// TwinCAT 3 PLC project Emulator
// ProgramVersion: 3.1.4024.12
// libraries:
//   Tc2_ModbusRTU, * (Beckhoff Automation GmbH)
//   Tc2_ModbusSrv, * (Beckhoff Automation GmbH)
//   Tc2_Standard, * (Beckhoff Automation GmbH)
//   Tc2_System, * (Beckhoff Automation GmbH)
//   Tc2_TcpIp, * (Beckhoff Automation GmbH)
//   Tc2_Utilities, * (Beckhoff Automation GmbH)
//   Tc3_Module, * (Beckhoff Automation GmbH)
// project tree:
//   00_FunctionsBlocks/AlarmManagement/ FB_AlarmCodeManager.TcPOU, FB_CheckCommand.TcPOU, FB_CheckSetpt.TcPOU, FB_DetectFixedValue.TcPOU, FB_DetectFlicker.TcPOU, FB_HeartBeatMasterBackup.TcPOU, FB_UnknownEvent.TcPOU, FUN_Alarms_CSV.TcPOU, FUN_ReadAlarm_CSV.TcPOU, ServerCSV.TcDUT, ServerSms.TcDUT, SMS_Server.TcPOU
//   00_FunctionsBlocks/Annexesfunction/ FUN_ConnectVPN.TcPOU, FUN_DisconnectVPN.TcPOU, FUN_GetPublicIp.TcPOU, FUN_PingHost.TcPOU, PRG_RestartPlc.TcPOU, PRG_RestartService.TcPOU
//   00_FunctionsBlocks/BoolManagement/ FB_CountNinTimeWindow.TcPOU, FB_TapVariable.TcPOU, FB_Toggle2Tap.TcPOU, FB_WordToArrayOfBool.TcPOU, FB_WriteOnChange.TcPOU, RS_NoReset.TcPOU
//   00_FunctionsBlocks/Communication/IEC104/ E_ComState.TcDUT, FB_IEC104ServerAkuo.TcPOU, GVL_Cst.TcGVL, ST_IEC104AkuoParam.TcDUT
//   00_FunctionsBlocks/Communication/Mail/ FUN_SendMail.TcPOU, ServerMail.TcDUT
//   00_FunctionsBlocks/Communication/ModbusRTU/ CheckStruct.TcPOU, FB_ModbusRTU.TcPOU, FB_ReadModbusRTU_V2.TcPOU, Sample_ModbusRTU.TcPOU, Struct_InputRTU.TcDUT
//   00_FunctionsBlocks/Communication/ModbusTCP/ FB_ModbusRead.TcPOU, FB_ModbusReadCoils.TcPOU, FB_ModbusReadInput.TcPOU, FB_ModbusReadInputRegs.TcPOU, FB_ModbusWrite.TcPOU, FB_ModbusWriteMultipleCoils.TcPOU, FB_ModbusWriteSingleCoil.TcPOU, FB_ModbusWriteSingleRegister.TcPOU
//   00_FunctionsBlocks/Communication/SMS/ FB_DeleteAllSMS.TcPOU, FB_DeleteSMS.TcPOU, FB_Extract_Num_Mes.TcPOU, FB_Login.TcPOU, FB_ReadSMS.TcPOU, FB_SendSMS.TcPOU, ST_SMSDataSetEntry_Read.TcDUT, ST_SMSDataSetEntry_Send.TcDUT
//   00_FunctionsBlocks/Ctrl/ FB_PIDRegulation.TcPOU
//   00_FunctionsBlocks/Database/ CheckConfig.TcPOU, PRG_EpochConverter.TcPOU, PRG_TimestructConverter.TcPOU, St_DataHisto.TcDUT, St_DataHisto_Epoch.TcDUT, UnixTimestamp.TcPOU
//   00_FunctionsBlocks/Database/Firebird/ Firebird_CreateTables.TcPOU, Firebird_InsertBuffer.TcPOU, Firebird_InsertBuffer_vEpoch.TcPOU, Firebird_ReadAlarms.TcPOU, Firebird_RetrieveHDBID.TcPOU, Firebird_SelectBuffer.TcPOU, Firebird_WriteAlarms.TcPOU, LoggerFirebird.TcDUT, St_AlarmsV2.TcDUT
//   00_FunctionsBlocks/Database/InfluxDb/ InfluxDb_AlarmsManagement.TcPOU, InfluxDb_ReadValues.TcPOU, InfluxDb_WriteAlarms.TcPOU, InfluxDb_WriteStruct.TcPOU, LoggerInfluxDb.TcDUT, ST_InfluxAlarmsInsert.TcDUT, ST_InfluxAlarmsRetrieve.TcDUT
//   00_FunctionsBlocks/Database/SQLCe/ FB_SQLExpert_InsertBuffer_1.TcPOU
//   00_FunctionsBlocks/Database/SQLite/ SQLite_CreateDb_V2_1.TcPOU, SQLite_DeleteConfDb_1.TcPOU
//   00_FunctionsBlocks/DataProcessing/Compress/ FB_CompressFile.TcPOU, FUN_CompressCSV.TcPOU
//   00_FunctionsBlocks/DataProcessing/Database/ DataBase_V2.TcPOU, FB_DeleteFile.TcPOU, FB_SQLExpert_InsertBuffer.TcPOU, SQLite_CreateDb_V2.TcPOU, SQLite_DeleteConfDb.TcPOU
//   00_FunctionsBlocks/DataProcessing/ FB_Average.TcPOU, FB_CountBitOfWordAtTrue.TcPOU, FB_Integrate.TcPOU, FB_MessageDynamique.TcPOU, FB_MovingAverage.TcPOU, FB_Ramp.TcPOU, FB_Ramp_Time.TcPOU, FB_Smooth.TcPOU, FB_XorWord.TcPOU, FUN_Transpose.TcPOU, ReplaceAll.TcPOU, SavePersistent.TcPOU, Split.TcPOU, Substring.TcPOU
//   00_FunctionsBlocks/DataProcessing/MergeWord/ FB_ISKRA_T5.TcPOU, FB_ISKRA_T6.TcPOU, FB_MergeWordsToDint.TcPOU, FB_MergeWordsToFloat.TcPOU, FB_MergeWordsToUint.TcPOU, FB_MergeWordsToUlint.TcPOU, FB_SplitFloatToWords.TcPOU, FB_WordsToDint64BE.TcPOU, FB_WordsToFloat32MLE.TcPOU
//   00_FunctionsBlocks/DataProcessing/ReadFile/ FB_Read.TcPOU, FB_ReadCSV.TcPOU
//   00_FunctionsBlocks/DataProcessing/SplitWord/ FB_SplitRealToWords.TcPOU, FB_SplitRealToWords_IEEE754.TcPOU, FB_SplitUlintToWords.TcPOU, FB_SplitWordToByte.TcPOU
//   00_FunctionsBlocks/DataProcessing/WriteFile/ CheckStruct_Alarms.TcPOU, FB_CreateDir_V2.TcPOU, FB_WriteFile.TcPOU, FB_Write_CSV.TcPOU, FUN_CreateDir_CSV.TcPOU, LoggerCSV.TcDUT, ST_Journal.TcDUT, ST_ValuesAlarms.TcDUT, ST_ValuesWrite.TcDUT
//   00_FunctionsBlocks/Fifo/ FB_CommandAlternate.TcPOU, FB_DBDatasetFifo.TcPOU, FB_DBDatasetFifo_1min.TcPOU, FB_SMSDatasetFifo_Read.TcPOU, FB_SMSDatasetFifo_Send.TcPOU, GVL_Fifo.TcGVL
//   00_FunctionsBlocks/HistorizationVisu/ FB_OperationIndex.TcPOU, GetTime.TcPOU
//   00_FunctionsBlocks/Templates/ FB_EX_Example.TcPOU
//   01_Equipement_Library/Actuators/ CB_AuxMVCB_Sch.TcDUT, CB.TcDUT, CB_Standard.TcDUT, FB_CB_AuxMVCB.TcPOU, FB_CB_Base.TcPOU, FB_CB_FeederMVCB.TcPOU, FB_CB_GridMVCB.TcPOU, FB_CB_MainHVCB.TcPOU, FB_CB_MainMVCB.TcPOU, FB_CB_MeasureMVCB.TcPOU, FB_CB_MVSwitch.TcPOU, CB_FeederMVCB_Sch.TcDUT, CB_MainHVCB_Sch.TcDUT, CB_MainMVCB_Sch.TcDUT, CB_MeasureMVCB_Sch.TcDUT
//   01_Equipement_Library/Batteries/ Cell.TcDUT, FB_SystemBMS_Base.TcPOU, FB_SystemBMS_M3.TcPOU, Rack.TcDUT, RackString.TcDUT, SystemBMS.TcDUT
//   01_Equipement_Library/Datalogger/ Datalogger.TcDUT, Datalogger_PPCVerrerie.TcDUT, Datalogger_SchSkid.TcDUT, Datalogger_SENECA.TcDUT, FB_Datalogger_Base.TcPOU, FB_Datalogger_PPCVerrerie.TcPOU, FB_Datalogger_SchSkid.TcPOU, FB_Datalogger_SENECA.TcPOU
//   01_Equipement_Library/Fan/ Fan.TcDUT, FB_Fan_Basic.TcPOU
//   01_Equipement_Library/FireSystem %28FSS%29/ FB_FSS.TcPOU (not stored), FSS.TcDUT (not stored), FSS_Standard.TcDUT (not stored)
//   01_Equipement_Library/GRID/ FB_GRID_Base.TcPOU, FB_GRID_Enedis.TcPOU, GRID.TcDUT, GRID_Enedis.TcDUT
//   01_Equipement_Library/HVAC/ FB_HVAC.TcPOU, FB_HVAC_Base.TcPOU, FB_HVAC_MADI.TcPOU, FB_HVAC_Standard.TcPOU, HVAC.TcDUT, HVAC_MADI.TcDUT, HVAC_Standard.TcDUT
//   01_Equipement_Library/Inverter/ FB_INV_1000CP_XT.TcPOU, FB_INV_Base.TcPOU, FB_INV_Sch4400.TcPOU, FB_INV_Smartlogger.TcPOU, FB_INV_Sun2000KtlMo.TcPOU, INV.TcDUT, INV_1000CP_XT.TcDUT, INV_1000CP_XT_StringMonitor.TcDUT, INV_Huawei.TcDUT, INV_Sch4400.TcDUT, SL_Huawei.TcDUT, STR.TcDUT
//   01_Equipement_Library/IPC/ FB_IPC.TcPOU, IPC.TcDUT
//   01_Equipement_Library/Operation Meter/ FB_PM_520_230.TcPOU, FB_PM_A40.TcPOU, FB_PM_Base.TcPOU, FB_PM_ION7650.TcPOU, FB_PM_Janitza.TcPOU, FB_PM_PM3250.TcPOU, FB_PM_PM800.TcPOU, FB_PM_SicamQ100.TcPOU, FB_PM_SM103E.TcPOU, PM.TcDUT, PM_PM800.TcDUT, PM_Q100.TcDUT, PM_SicamQ100.TcDUT, PM_Standard.TcDUT
//   01_Equipement_Library/PCS/ FB_PCS_Base.TcPOU, FB_PCS_Jema.TcPOU, PCS.TcDUT, PowerCol_Jema.TcDUT, PowerCol_Jema_Alarms.TcDUT
//   01_Equipement_Library/ProtectRelay/ FB_ProtectRelay_Base.TcPOU, FB_ProtectRelay_DM2.TcPOU, FB_ProtectRelay_Flair23DM.TcPOU, FB_ProtectRelay_NSXCB.TcPOU, FB_ProtectRelay_PACE100ST.TcPOU, FB_ProtectRelay_REF615.TcPOU, FB_ProtectRelay_SEPAM10a.TcPOU, FB_ProtectRelay_SepamS48.TcPOU, FB_ProtectRelay_SepamT20.TcPOU, FB_ProtectRelay_VIP410.TcPOU, FB_ProtectRelay_WIP1.TcPOU, ProtectRelay.TcDUT, ProtectRelay_Flair23DM.TcDUT, ProtectRelay_NSXCB.TcDUT, ProtectRelay_PACE100ST.TcDUT, ProtectRelay_REFIO.TcDUT, ProtectRelay_S42.TcDUT, ProtectRelay_S48.TcDUT, ProtectRelay_T20.TcDUT, ProtectRelay_T87.TcDUT, ProtectRelay_VIP410.TcDUT, ProtectRelay_WIP1.TcDUT
//   01_Equipement_Library/Router/ FB_Router.TcPOU, Router.TcDUT, Router_Standard.TcDUT
//   01_Equipement_Library/Sensors/ANA/ ANA.TcDUT, FB_ANA_Base.TcPOU, FB_ANA_IO.TcPOU, FB_ANA_Irra_Fx.TcPOU
//   01_Equipement_Library/Sensors/COM/ AllInOne.TcDUT, FB_AllInOne.TcPOU, FB_ANA_SMP1X.TcPOU, SMP1X.TcDUT
//   01_Equipement_Library/Sensors/TOR/ FB_TOR_Base.TcPOU, FB_TOR_CB.TcPOU, FB_TOR_DS.TcPOU, FB_TOR_ES.TcPOU, FB_TOR_Fuse.TcPOU, FB_TOR_MS.TcPOU, FB_TOR_Rain.TcPOU, FB_TOR_SD.TcPOU, FB_TOR_Spd.TcPOU, FB_TOR_Standard.TcPOU, FB_TOR_ToS.TcPOU, TOR.TcDUT, TOR_Rain.TcDUT, TOR_Standard.TcDUT
//   01_Equipement_Library/Tariff Meter/ EM.TcDUT, EM_Standard.TcDUT, FB_EM.TcPOU, FB_EM_Base.TcPOU, FB_EM_Pulse.TcPOU
//   01_Equipement_Library/Transfo/ FB_Transfo_Base.TcPOU, FB_Transfo_HVCom.TcPOU, FB_Transfo_MV.TcPOU, FB_Transfo_MVCom.TcPOU, Transfo.TcDUT, Transfo_HV.TcDUT, Transfo_MV.TcDUT
//   01_Equipement_Library/UPS/ FB_UPS_Base.TcPOU, FB_UPS_CXC.TcPOU, FB_UPS_Eneris.TcPOU, FB_UPS_PS10048.TcPOU, UPS.TcDUT, UPS_CXC.TcDUT, UPS_ENERIS.TcDUT, UPS_Eneris.TcDUT, UPS_Eneris.TcDUT, UPS_PS10048.TcDUT
//   02_Product_Library/EnergyStorageSystem%28ESS%29/ ESS.TcDUT (not stored), FB_ESS.TcPOU (not stored), FB_ESS_Base.TcPOU (not stored)
//   02_Product_Library/PowerTRansformerStation%28PTR%29/ FB_PTR.TcPOU (not stored), FB_PTR_Base.TcPOU (not stored), PTR.TcDUT (not stored), PTR_Exd.TcDUT (not stored)
//   02_Product_Library/Substation%28SUB_HV%29/ FB_SUBHV.TcPOU (not stored), FB_SUBHV_Base.TcPOU (not stored), SUBHV.TcDUT (not stored), SUBHV_Exd.TcDUT (not stored)
//   02_Product_Library/Substation%28SUB_MV%29/ FB_SUBMV.TcPOU (not stored), FB_SUBMV_Base.TcPOU (not stored), SUBMV.TcDUT (not stored), SUBMV_Exd.TcDUT (not stored)
//   02_Product_Library/WeatherStation %28WS%29/ FB_WS.TcPOU (not stored), FB_WS_Base.TcPOU (not stored), WS.TcDUT (not stored), WS_AGMA.TcDUT (not stored)
//   03_Power_Plant %28PP%29/ FB_PP.TcPOU (not stored), PP.TcDUT (not stored)
//   04_Application/ADS/ ADS_Custom.TcPOU, ADS_Param.TcPOU
//   04_Application/Checks/ CheckBounds.TcPOU, CheckDivDInt.TcPOU, CheckDivLInt.TcPOU, CheckDivLReal.TcPOU, CheckDivReal.TcPOU, CheckLRangeSigned.TcPOU, CheckLRangeUnsigned.TcPOU, CheckPointer.TcPOU, CheckRangeSigned.TcPOU, CheckRangeUnsigned.TcPOU
//   04_Application/CONFIG/ GVL_BASE.TcGVL, GVL_Beckhoff.TcGVL, GVL_CFG.TcGVL, GVL_Check.TcGVL, GVL_DataBaseStructures.TcGVL, GVL_EmulConfig.TcGVL
//   04_Application/IO/ IO.TcDUT, PRG_IO.TcPOU, ST_AI.TcDUT, ST_AO.TcDUT, ST_DI.TcDUT, ST_DO.TcDUT
//   04_Application/MAIN/ MAIN_Emul.TcPOU
//   / Emul_Task.TcTTO

CONFIGURATION Emulator
    RESOURCE PLC ON TwinCAT3
        TASK Emul_Task(INTERVAL := T#25000us, PRIORITY := 16);
        PROGRAM MAIN_Emul WITH Emul_Task : MAIN_Emul;
    END_RESOURCE
END_CONFIGURATION

// ---- 00_FunctionsBlocks/AlarmManagement/ServerCSV.TcDUT

TYPE ServerCSV :
STRUCT
	FileSize			: ULINT;			(*(o) Size of the file being used for logging alarms *)
	TimeCreation		: TIMESTRUCT;		(* TimeCreation of file*)
	TimeModif			: TIMESTRUCT;		(* Time Modif of file*)
	MesAlarmCode		: WORD;				(* Alarm Code related to this functionnality*)

END_STRUCT
END_TYPE

// ---- 00_FunctionsBlocks/AlarmManagement/ServerSms.TcDUT

TYPE ServerSms :
STRUCT
	NbrUtiliActive			: INT;									(* Number of users*)
	MesAlarmCode			: WORD;									(* Alarm Code*)
	AX_Numtel				: ARRAY[1..CstNbUser] OF STRING(26);	(*Tel Number list*)
	AX_Subscribed			: ARRAY[1..CstNbUser] OF BOOL;			(*Subscription list*)
	AX_NomUtili				: ARRAY[1..CstNbUser] OF STRING(50); 	(* User name list	*)
	AX_UserLVL				: ARRAY[1..CstNbUser] OF WORD; 		(*User Level*)

END_STRUCT
END_TYPE

// ---- 00_FunctionsBlocks/Communication/IEC104/E_ComState.TcDUT
TYPE E_ComState :
(
	INIT := 0,
	IDLE,
	CONNECT,
	DATATRANSFER,
	DISCONNECT
);
END_TYPE

// ---- 00_FunctionsBlocks/Communication/IEC104/ST_IEC104AkuoParam.TcDUT
TYPE ST_IEC104AkuoParam :
STRUCT
	bEnableFlicker 	: BOOL :=  TRUE ;
	tFlickerWindow	: TIME := T#10S ; 
	uFlickerNumber	: UINT := 7  ; 

	iLocalPort 		: UDINT := 2404;						// locl port
	sLocalHost		: STRING := '127.0.0.1'; 			// server IP address. 
	iAOnb			: INT ;								// Number of AO being treated ( <GVL_Cst.CstNbAOEntries)
 
END_STRUCT
END_TYPE

// ---- 00_FunctionsBlocks/Communication/Mail/ServerMail.TcDUT

TYPE ServerMail :
STRUCT

	MesAlarmCode			: WORD;			(*alarm code *)
	
	AX_MailAddr				: ARRAY[1..CstNbUser] OF STRING(255);		(* Mail Address List*)
	AX_Subscribed			: ARRAY[1..CstNbUser] OF BOOL;				(* Mail subscription list*)
	AX_NomUtili				: ARRAY[1..CstNbUser] OF STRING(50); 		(* User Name List*)
	AX_UserLVL				: ARRAY[1..CstNbUser] OF WORD; 		(* User Level*)
	
	OUT_NbMailSent			: ULINT;									(* Number of mail being sent *)
	
END_STRUCT
END_TYPE

// ---- 00_FunctionsBlocks/Communication/ModbusRTU/Struct_InputRTU.TcDUT
TYPE Struct_InputRTU :
STRUCT
	InStartAddr			: WORD;
	InQuantity			: WORD;
	InUnitID			: BYTE;
	InBuffer			: POINTER TO BYTE;
	InFunction			: UINT;
	OutBusy				: POINTER TO BOOL;
	OutError			: POINTER TO BOOL;
	OutCompleted 		: POINTER TO BOOL;
	OutErrorId			: POINTER TO INT ; 
END_STRUCT
END_TYPE

// ---- 00_FunctionsBlocks/Communication/SMS/ST_SMSDataSetEntry_Read.TcDUT
TYPE ST_SMSDataSetEntry_Read :
STRUCT
	Message : STRING(160);  // Commande envoyé par message
	Num		: STRING(20);  //  Numéro de l'utilisateur
END_STRUCT
END_TYPE

// ---- 00_FunctionsBlocks/Communication/SMS/ST_SMSDataSetEntry_Send.TcDUT
TYPE ST_SMSDataSetEntry_Send :
STRUCT
	ID				: UINT;			// Unic ID to identify the alarm
	IndexWord		: UINT; 		//Index du word correspondant aux alarmes
	IndexBit		: UINT; 		//Index du bit correspondant a l'alarme
	Active			: BOOL; 		//Ne pas remplir - Utilisé par le code
	Num_tel			: STRING(20);//Ne pas remplir - Utilisé par le code
	TimeStamp_Act	: STRING;	// TimeStamp of the last activation or desactivation
	Alarms_LVL		: WORD;
END_STRUCT
END_TYPE

// ---- 00_FunctionsBlocks/Database/Firebird/LoggerFirebird.TcDUT

TYPE LoggerFirebird :
STRUCT
	MesAlarmCode		: WORD;				// Alarm Code

END_STRUCT
END_TYPE

// ---- 00_FunctionsBlocks/Database/Firebird/St_AlarmsV2.TcDUT
TYPE St_AlarmsV2 :
STRUCT
	TIMESTAMP_START : DT;
	TIMESTAMP_STOP	: DT;
	ALARMSID 		: DINT;
	ACT				: INT;
	ACK				: INT;
	

END_STRUCT
END_TYPE

// ---- 00_FunctionsBlocks/Database/InfluxDb/LoggerInfluxDb.TcDUT
TYPE LoggerInfluxDb :
STRUCT
	MesAlarmCode		: WORD;				// Alarm Code
END_STRUCT
END_TYPE

// ---- 00_FunctionsBlocks/Database/InfluxDb/ST_InfluxAlarmsInsert.TcDUT
TYPE ST_InfluxAlarmsInsert :
STRUCT
    {attribute 'TagName' := 'Message'}
	Message		 	: T_MaxString;	// Alarm Message 
    {attribute 'FieldName' := 'ID'}	
	ID			: 	ULINT;
    {attribute 'FieldName' := 'Value'}	
	Value 		: BOOL;
    {attribute 'FieldName' := 'Ack'}	
	Ack			: BOOL;	
END_STRUCT
END_TYPE

// ---- 00_FunctionsBlocks/Database/InfluxDb/ST_InfluxAlarmsRetrieve.TcDUT
TYPE ST_InfluxAlarmsRetrieve :
STRUCT
    {attribute 'TagName' := 'time'}
	MesTime			: LINT;
    {attribute 'TagName' := 'Message'}
	Message		 	: T_MaxString;	// Alarm Message 
    {attribute 'FieldName' := 'ID'}	
	ID				: ULINT;
    {attribute 'FieldName' := 'Value'}	
	Value 			: BOOL;
    {attribute 'FieldName' := 'Ack'}	
	Ack				: BOOL;	
END_STRUCT
END_TYPE

// ---- 00_FunctionsBlocks/Database/St_DataHisto.TcDUT
TYPE St_DataHisto :
STRUCT
	Timestamp		: TIMESTRUCT;
	ParentId		: DINT;
	Value			: LREAL;
END_STRUCT
END_TYPE

// ---- 00_FunctionsBlocks/Database/St_DataHisto_Epoch.TcDUT
TYPE St_DataHisto_Epoch :
STRUCT
	Timestamp		: ULINT;
	ParentId		: DINT;
	Value			: LREAL;
END_STRUCT
END_TYPE

// ---- 00_FunctionsBlocks/DataProcessing/WriteFile/LoggerCSV.TcDUT

TYPE LoggerCSV :
STRUCT
	FileSize			: ULINT;			(* (o) File size *)
	TimeCreation		: TIMESTRUCT;		(* TimeCreation of file*)
	TimeModif			: TIMESTRUCT;		(* Time Modif of file*)
	MesAlarmCode		: WORD;				(* Alarm Code*)

END_STRUCT
END_TYPE

// ---- 00_FunctionsBlocks/DataProcessing/WriteFile/ST_Journal.TcDUT
TYPE ST_Journal :
STRUCT
	Message			: STRING(150); //Message texte à envoyer aux utilisateurs
	Groupe			: (Sans_Operation,Avec_Operation_Act,Avec_Operation_Act_Des):=1; // 0:sans action,1:Envois sms sur acttivation,2:Envois sms sur activation et desactivation
	Ax_ParamB		: ARRAY [1..4] OF POINTER TO BOOL; //Tableau boolean permettant d'envoyer un message dynamique.
	Ax_ParamI		: ARRAY [1..4] OF POINTER TO SINT; //Tableau Sint permettant d'envoyer un message dynamique.
END_STRUCT
END_TYPE

// ---- 00_FunctionsBlocks/DataProcessing/WriteFile/ST_ValuesAlarms.TcDUT
TYPE ST_ValuesAlarms :
STRUCT
	ID				: UINT;		// Unic ID to identify the alarm 
	Message		 	: STRING(160);	// Alarm Message 
	Value 			: BOOL;		// Value of the alarm
	Ack 			: BOOL;		// Ack of the alarm	
	TimeStamp_Act	: STRING;	// TimeStamp of the last activation or desactivation
	
	Groupe			: UINT:=0; // 0:sans action,1:Envois sms sur acttivation,2:Envois sms sur activation et desactivation
	Alarms_LVL		: WORD:=1; // Si Num utilisateur > Alarms_LVL alors il ne recoit pas les sms 1 := Standart , 2 := Syntehses , 3:= Securité
END_STRUCT
END_TYPE

// ---- 00_FunctionsBlocks/DataProcessing/WriteFile/ST_ValuesWrite.TcDUT
TYPE ST_ValuesWrite :
STRUCT
	Description : STRING;
	Address 	: POINTER TO REAL;
	AddressLR	: POINTER TO LREAL;
	AddressUL	: POINTER TO ULINT;
	AddressUI	: POINTER TO UINT;
	Size		: UINT;
	Sampling	: DINT := 1000;		// Period of sampling
	
END_STRUCT
END_TYPE

// ---- 01_Equipement_Library/Actuators/CB_AuxMVCB_Sch.TcDUT
///////////
// Structure For Bousquet. Main Operating Data to be saved (ex: OPC).  
//////////

TYPE CB_AuxMVCB_Sch :
STRUCT
	//DI
	MesData					: CB ;      (* Object*)
	MesFuseBurned		    : BOOL ; 	(* The Fuse is burned*)
	MesEarth				: BOOL ; 	(* The Cell is grounded*)

END_STRUCT
END_TYPE

// ---- 01_Equipement_Library/Actuators/CB.TcDUT
TYPE CB :
///////////
// Structure For Bousquet. Main Operating Data to be saved ( ex: OPC )   
//////////
STRUCT
	//DI
	MesClosed		: BOOL ;	(* Cell is closed*)
	MesOpened		: BOOL ;	(* cell is opened*)
	
	MesAlarmCode	: WORD ;	(* Internal Akuo Alarm Code*)
	MesWarningCode	: WORD ;	(* Internal Akuo Warning Code*)
	MesEventCode	: WORD ;	(* Internal Akuo Warning Code*)
	
	MesCP_Open		: BOOL ;   	(* Cal(NA) Permanent Conditions*)
	MesCP_Close		: BOOL ; 	(* Cal(NA) Permanent Conditions*) 

END_STRUCT
END_TYPE

// ---- 01_Equipement_Library/Actuators/CB_Standard.TcDUT
TYPE CB_Standard :
///////////
// Structure For Bousquet. Main Operating Data to be saved ( ex: OPC )   
//////////
STRUCT
	//DI
	MesData				: CB ;  (* Object*)

END_STRUCT
END_TYPE

// ---- 01_Equipement_Library/Actuators/CB_FeederMVCB_Sch.TcDUT
///////////
// Structure For Bousquet . Main Operating Data to be saved (ex: OPC).  
//////////

TYPE CB_FeederMVCB_Sch :
STRUCT
	//DI
	MesData					: CB   ;    (* Object*)
	MesComutLocal		    : BOOL ; 	(* The cell selector is in local position*)
	MesAlarmPwr		        : BOOL ; 	(* The cell motorization has a power supply fault*)
	MesEarth				: BOOL ; 	(* The cell is grounded (earthing)*)
	MesTripped	    	    : BOOL ; 	(* The cell is tripped (opened and locked due to alarm)*)
	OUT_CmdOpen				: BOOL ; 	(* The SCADA sends an Open command to the cell*)
	OUT_CmdClose			: BOOL ; 	(* The SCADA sends a Close command to the cell*)
	MesOpened_Sect			: BOOL ;    (* The associated switchgear is opened*)
	
END_STRUCT
END_TYPE

// ---- 01_Equipement_Library/Actuators/CB_MainHVCB_Sch.TcDUT
///////////
// Structure For Bousquet . Main Operating Data to be saved (ex: OPC).  
//////////

TYPE CB_MainHVCB_Sch :
STRUCT
	//DI
	MesData					: CB   ;    (* Object*)
	MesComutLocal		    : BOOL ; 	(* The cell selector is in local position*)
	MesAlarmPwr		        : BOOL ; 	(* The cell motorization has a power supply fault*)
	MesEarth				: BOOL ; 	(* The cell is grounded (earthing)*)
	MesTripped	    	    : BOOL ; 	(* The cell is tripped (opened and locked due to alarm)*)

	MesAlarm_SF6      			: BOOL ; (* Not enough SF6 gaz *)
	MesAlarm_Disarmed      		: BOOL ; (* HVCB Command is disarmed*)
	MesAlarm_ArmingMotor   		: BOOL ; (* Arming motorization is on fault*)
	MesAlarm_230V  		 		: BOOL ; (* 230V Aux is on fault*)
	MesOpened_Sect				: BOOL ; (* The associated switchgear is opened*)
	
END_STRUCT
END_TYPE

// ---- 01_Equipement_Library/Actuators/CB_MainMVCB_Sch.TcDUT
///////////
// Structure for MainMVCB Schneider. Main Operating Data to be saved (ex: OPC).  
//////////

TYPE CB_MainMVCB_Sch :
STRUCT
	//DI
	MesData					: CB   ;    (* Object*)
	MesComutLocal		    : BOOL ; 	(* The cell selector is in local position*)
	MesAlarmPwr		        : BOOL ; 	(* The cell motorization has a power supply fault*)
	MesEarth				: BOOL ; 	(* The cell is grounded (earthing)*)
	MesTripped	    	    : BOOL ; 	(* The cell is tripped (opened and locked due to alarm)*)
	OUT_CmdOpen				: BOOL ; 	(* The SCADA sends an Open command to the cell*)
	OUT_CmdClose			: BOOL ; 	(* The SCADA sends a Close command to the cell*)
	MesOpened_Sect			: BOOL ; 	(* The associated switchgear is opened*)
	
END_STRUCT
END_TYPE

// ---- 01_Equipement_Library/Actuators/CB_MeasureMVCB_Sch.TcDUT
///////////
// Structure For Bousquet. Main Operating Data to be saved (ex: OPC).  
//////////

TYPE CB_MeasureMVCB_Sch :
STRUCT
	//DI
	MesData					: CB ;      (* Object*)
	MesFuseBurned		    : BOOL ; 	(* The Fuse is burned*)
	MesEarth				: BOOL ; 	(* The Cell is grounded*)

END_STRUCT
END_TYPE

// ---- 01_Equipement_Library/Batteries/Cell.TcDUT
///////////
// Structure For Battery Racks. Main Operating Data to be saved ( ex: OPC ) .  
//////////
TYPE Cell :
STRUCT
	MesU			: REAL ;    		(*( V) Cell voltage *)
	
END_STRUCT
END_TYPE

// ---- 01_Equipement_Library/Batteries/Rack.TcDUT
///////////
// Structure For Battery Racks. Main Operating Data to be saved ( ex: OPC ) .  
//////////
TYPE Rack :
STRUCT
	
		// Info of Rack BBMS  
		ParamNbStrings			: UINT ; 	// 		Number of strings for the rack set in BBMS 
		MesHeartBeat			: UINT;		// (NA) Rack's Heartbeat, increases by 1 every second
		MesAlarm1				: WORD;		// (NA) bit0: 
		MesAlarm2				: WORD;		// (NA) bit0: 
		MesProtection1			: WORD;		// (NA) bit0: 
		MesProtection2			: WORD;		// (NA) bit0: 		
		MesSwitchControlStatus	: WORD ; 	// Control status
		MesSwitchSensorStatus	: WORD ; 	// Sensor status
		MesUSwtchGrPackPlus		: REAL;		// (V)	a measured value of voltage applied to pack(+) of switchgear
		MesTempPCB				: REAL ; 	// (°C) Temperature Rack PCB 
		MesIdcFaultLvl			: UINT ;	//		Current Level when power is cut (1/2/3/4/5/6/7/8/9/10 : 1200A/700A/500A/200A/0A/-0A/-200A/-500A/-700A/-1200A)
		MesDcOpenCount			: UINT ; 	// Count number of dc opening 
		MesDcCloseCount			: UINT ; 	// Count number of dc closing 
		
		AX_RACKSTRING			: ARRAY[1..1] OF RackString ; 	// object 
	
		CalRackClosed			: BOOL ; 		// Rack ( Main DC contactor )is closed 

END_STRUCT
END_TYPE

// ---- 01_Equipement_Library/Batteries/RackString.TcDUT
///////////
// Structure For Battery Racks. Main Operating Data to be saved ( ex: OPC ) .  
//////////
TYPE RackString :
STRUCT
	
		MesMode								: UINT;		// (NA) Rack mode: 0: None, 1: Init, 2: Off, DcSwitch On, 3: On, DcSwitch On,
		MesAlarm1							: WORD;		// (NA) bit0: 
		MesAlarm2							: WORD;		// (NA) bit0: 
		MesAlarm3							: WORD;		// (NA) bit0: 
		MesAlarm4							: WORD;		// (NA) bit0: 
		MesProtection1						: WORD;		// (NA) bit0: 
		MesProtection2						: WORD;		// (NA) bit0: 
		MesProtection3						: WORD;		// (NA) bit0: 
		MesProtection4						: WORD;		// (NA) bit0: 		
		MesControlStatus					: WORD ; 	// Control Status
		MesUdc								: REAL ; 	// String Voltage 
		MesUdc_ModuleSum					: REAL  ;	// String voltage obtained by summing module voltage 
		MesUdc_CellSum						: REAL ; 	// String voltage obtained by summing Cell voltage 
		MesIdc								: REAL;		// (A) Rack Current
		MesIdc_Avg							: REAL;		// (A) Rack Current ( average of 3 sec) 
		MesSoC	 							: REAL;  	// (%) SoC on Battery rack 
		MesSoH	 							: REAL;  	// (%) SoH on Battery rack 
		MesCCL								: REAL;		// (A) Charge limit of rack
		MesDCL								: REAL;		// (A) Discharge limit of rack
		MesCPL								: REAL ; 	// (kW) Charge Power Limit		- To zero if Estop is set . 
		MesDPL								: REAL ; 	// (kW) Discharge Power Limit - To zero if Estop is set .
		MesECharge							: REAL ; 	// (kWh) Total Energy charged over time 
		MesEDischarge						: REAL ; 	// (kWh) Total Energy Discharge over time 
		MesOff_ModuleID						: UINT; 	// Module ID where the power is off while the other modules are connected . 
		MesComError_ModuleID				: UINT ; 	// Module ID where there is a LOC while other modules are connected . 
		MesUdcDiffMax_Cell					: REAL ; 	// (V) 	Max voltage difference between cells . 
		MesUdc_Cell							: REAL; 	// (V)	Cell voltage. Average
		MesUdcMax1_Cell						: REAL; 	// (V)	Cell voltage. Max Rank #1
		MesUdcMax1_Cell_ModuleID			: UINT; 	// (V)	Module ID where Cell voltage  reaches Max value. Rank #1
		MesUdcMax1_Cell_CellID				: UINT; 	// (V)	Cell ID where Cell voltage reaches Max value. Rank #1
		MesUdcMin1_Cell						: REAL; 	// (V)	Cell voltage . Min Rank #1
		MesUdcMin1_Cell_ModuleID			: UINT; 	// (V)	Module ID where Cell voltage  reaches Min value. Rank #1
		MesUdcMin1_Cell_CellID				: UINT; 	// (V)	Cell ID where Cell voltage reaches Min value. Rank #1
		MesUdcMax2_Cell						: REAL; 	// (V)	Cell voltage . Max Rank #2
		MesUdcMax2_Cell_ModuleID			: UINT; 	// (V)	Module ID where Cell voltage  reaches Max value. Rank #2
		MesUdcMax2_Cell_CellID				: UINT; 	// (V)	Cell ID where Cell voltage reaches Max value. Rank #2
		MesUdcMin2_Cell						: REAL; 	// (V)	Cell voltage . Min Rank #2
		MesUdcMin2_Cell_ModuleID			: UINT; 	// (V)	Module ID where Cell voltage  reaches Min value. Rank #2
		MesUdcMin2_Cell_CellID				: UINT; 	// (V)	Cell ID where Cell voltage reaches Min value. Rank #2		
		MesTempDiffMax_Cell					: REAL ; 	// (°C) Max Temp difference between cells . 
		MesTemp_Cell						: REAL; 	// (°C)	Cell Temp . Average
		MesTempMax1_Cell					: REAL; 	// (°C)	Cell Temp . Max Rank #1
		MesTempMax1_Cell_ModuleID			: UINT; 	// (°C)	Module ID where Cell Temp  reaches Max value. Rank #1
		MesTempMax1_Cell_CellID				: UINT; 	// (°C)	Cell ID where Cell Temp reaches Max value. Rank #1
		MesTempMin1_Cell					: REAL; 	// (°C)	Cell Temp . Min Rank #1
		MesTempMin1_Cell_ModuleID			: UINT; 	// (°C)	Module ID where Cell Temp  reaches Min value. Rank #1
		MesTempMin1_Cell_CellID				: UINT; 	// (°C)	Cell ID where Cell Temp reaches Min value. Rank #1
		MesTempMax2_Cell					: REAL; 	// (°C)	Cell Temp . Max Rank #2
		MesTempMax2_Cell_ModuleID			: UINT; 	// (°C)	Module ID where Cell Temp  reaches Max value. Rank #2
		MesTempMax2_Cell_CellID				: UINT; 	// (°C)	Cell ID where Cell Temp reaches Max value. Rank #2
		MesTempMin2_Cell					: REAL; 	// (°C)	Cell Temp . Min Rank #2
		MesTempMin2_Cell_ModuleID			: UINT; 	// (°C)	Module ID where Cell Temp  reaches Min value. Rank #2
		MesTempMin2_Cell_CellID				: UINT; 	// (°C)	Cell ID where Cell Temp reaches Min value. Rank #2		
		MesTempPCBMax						: REAL ; 	// (°C) Temperature PCB Max
		MesTempPCBMax_ModuleID				: UINT ;    // (°C) Temperature PCB Max module ID
		MesTempPCBMin						: REAL ;    // (°C) Temperature PCB Min
		MesTempPCBMin_ModuleID				: UINT ; 	// (°C) Temperature PCB Min Module ID 	
		MesSensorStatus						: UINT ; 	//	Register status (only for Samsung diagnosis)
		MesModuleScanStatus					: UINT ; 	//	Register status (only for Samsung diagnosis)
		MesModuleBalancingStatus			: UINT ; 	//	Register status (only for Samsung diagnosis)
		MesModuleAddressStatus				: UINT ; 	//	Register status (only for Samsung diagnosis)
		MesModuleVoltageStatus				: UINT ; 	//	Register status (only for Samsung diagnosis)	
		MesModuleTemperatureStatus			: UINT ; 	//	Register status (only for Samsung diagnosis)
		MesUdcDiffCellMax					: REAL ; 	// (V)[Rack#1][String#1] Difference Voltage (MAX(Cell Sensing Summation))
		MesUdcDiffModuleMax					: REAL ; 	// (V)[Rack#1][String#1] Difference Voltage (Max(Module Sensing))        
		MesUdcDiffModuleMax_ModuleID		: UINT ; 	// [Rack#1][String#1] Difference Voltage (Max) Module Position           
		MesUdcDiffCellMin					: REAL ; 	// (V)[Rack#1][String#1] Difference Voltage (Min(Cell Sensing Summation))
		MesUdcDiffModuleMin					: REAL ; 	// (V)[Rack#1][String#1] Difference Voltage (Min(Module Sensing))        
		MesUdcDiffModuleMin_ModuleID		: UINT ; 	// [Rack#1][String#1] Difference Voltage (Min) Module Position           
		MesState							: UINT ; 	// internal string state machine . 
		MesCellVDist_under20mV				: REAL ; 	// (%)[Rack#1][String#1] Cell V Distribution (Under 20mV)
		MesCellVDist_underVimbAlarm 		: REAL ; 	// (%)[Rack#1][String#1] Cell V Distribution (Under V-IMB Alarm Level)
		MesCellVDist_underVimbProtection 	: REAL ; 	// (%)[Rack#1][String#1] Cell V Distribution (Under V-IMB Protection Level)
		MesCellVDist_VimbProtection 		: REAL ; 	// (%)[Rack#1][String#1] Cell V Distribution (V-IMB Protection Level or More)
		MesCellBalancingCntMax				: UINT ; 	// ()[Rack#1][String#1] Cell Balancing Execution Count (Max)
		MesCellBalancingCntMax_ModuleID		: UINT ; 	// ()[Rack#1][String#1] Cell Balancing Execution Count (Max) Module Position
		MesCellBalancingCntMax_CellID		: UINT ; 	// ()[Rack#1][String#1] Cell Balancing Execution Count (Max) Cell Position
		MesMaxBalancingTime					: REAL ; 	// (min)[Rack#1][String#1] Max Balancing Time (minute)
		
	
END_STRUCT
END_TYPE

// ---- 01_Equipement_Library/Batteries/SystemBMS.TcDUT
///////////
// Structure For Battery Controller. Main Operating Data to be saved ( ex: OPC ) .  
//////////

TYPE SystemBMS :
STRUCT
	
	MesHeartBeat				: UINT;			(* (NA) Goes from 0 to 999 every s*)
	MesNbRackConnected			: UINT;			(* (NA) Nb of Racks in service ( strings )*)
	MesNbRackTot				: UINT;			(* (NA) Total Nb of Racks (strings )*)
	MesIdcConnected				: REAL;			(* (A) Summation of all racks*)
	MesUdcConnected				: REAL;			(* (V) Voltage connected 	( average )*)
	MesUdcConnectedMedian		: REAL;			(* (V) Voltage connected 	( median )*)
	MesUdcConnectedMax			: REAL;			(* (V) Voltage connected 	( max )*)
	MesUdcConnectedMin			: REAL;			(* (V) Voltage connected 	( min )*)
	MesSoCConnected				: REAL; 		(* (%) SoC average ( priority : 1 if one is 0 all are 0  , 2 : one is 100 all are 100 , 3 : average )*)
	MesSoCConnectedMedian		: REAL; 		(* (%) SoC median value*)
	MesSoCConnectedMax			: REAL; 		(* (%) SoC Max value*)
	MesSoCConnectedMin			: REAL; 		(* (%) SoC Min value*)
	MesIdc						: REAL;			(* (A) Summation of all racks*)
	MesUdc						: REAL;			(* (V) Voltage of the rack, average*)
	MesUdcMedian				: REAL;			(* (V) Voltage of the rack, median*)
	MesUdcMax					: REAL;			(* (V) Voltage of the rack, max*)
	MesUdcMin					: REAL;			(* (V) Voltage of the rack, min*)
	MesSoC						: REAL; 		(* (%) SoC Average (not including racks with protection ) .*)
	MesSoCMedian				: REAL; 		(* (%) SoC Median*)
	MesSoCMax					: REAL; 		(* (%) SoC Max*)
	MesSoCMin					: REAL; 		(* (%) SoC Min*)
	MesSoH						: REAL; 		(* (%) SoH Average*)
	MesSoHMedian				: REAL; 		(* (%) SoH Median*)
	MesSoHMax					: REAL; 		(* (%) SoH Max*)
	MesSoHMin					: REAL; 		(* (%) SoH Min*)
	MesUdc_Cell					: REAL; 		(* (V)  Cell voltage among all strings in system. Average*)
	MesUdcMedian_Cell			: REAL; 		(* (V)  Cell voltage among all strings in system. Median*)
	MesUdcMax_Cell				: REAL; 		(* (V)Cell voltage among all strings in system. Max*)
	MesUdcMax_Cell_RackID		: UINT:=1 ; 	(* (V)Rack ID where Cell voltage among all strings in system reaches Max value.*)
	MesUdcMin_Cell				: REAL; 		(* (V) Cell voltage among all strings in system. Min*)
	MesUdcMin_Cell_RackID		: UINT :=1 ; 	(* (V)Rack ID where Cell voltage among all strings in system reaches Min value.*)
	MesUdcDiffMax_Cell			: REAL; 		(* (V) Max Cell voltage difference among all strings in system. Min*)
	MesUdcDiffMax_Cell_RackID	: UINT:=1 ; 	(* (V)Rack ID where Cell voltage among all strings in system reaches Min value.*)
	MesTmp_Cell					: REAL; 		(* (°C)  Cell Temperature among all strings in system. Average*)
	MesTmpMedian_Cell			: REAL; 		(* (°C)  Cell Temperature among all strings in system. Median*)
	MesTmpMax_Cell				: REAL; 		(* (°C)Cell Temperature among all strings in system. Max*)
	MesTmpMax_Cell_RackID		: UINT:=1 ; 	(* (°C)Rack ID where Cell Temperature among all strings in system reaches Max value.*)
	MesTmpMin_Cell				: REAL; 		(* (°C) Cell Temperature among all strings in system. Min*)
	MesTmpMin_Cell_RackID		: UINT:=1 ; 	(* (°C)Rack ID where Cell Temperature among all strings in system reaches Min value.*)
	MesTmpDiffMax_Cell			: REAL; 		(* (°C) Max Cell Temperature difference among all strings in system.*)
	MesTmpDiffMax_Cell_RackID	: UINT:=1 ; 	(* (°C)Rack ID where Cell Temperature among all strings in system reaches Max diff value*)
	MesCCL						: REAL;			(* (A) Charge Current Limit*)
	MesDCL						: REAL;			(* (A) Discharge Current Limit*)
	MesCPL						: REAL ; 		(* (kW) Charge Power Limit		- To zero if Estop is set .*)
	MesDPL						: REAL ; 		(* (kW) Discharge Power Limit - To zero if Estop is set .*)
	MesECharge					: REAL ; 		(* (kWh) 	Total Energy charged over time*)
	MesEDischarge				: REAL ; 		(* (kWh)	Total Energy Discharge over time*)
	MesWatchdog					: WORD;			(* (NA) Inverses the WatchdogQuery*)
	MesUdc_PartialOp			: REAL ; 		(* (V) Voltage of the Rack with the highest number of strings which are under Partial Op due to limit of voltage difference alarm*)
	MesUdc_PartialOp_RackID		: UINT :=1 ; 	(* (V) Rack ID where Voltage of the Rack with the highest number of strings which are under Partial Op due to limit of voltage difference alarm*)
	MesUdc_PartialOp_StringID	: UINT :=1 ; 	(* (V) Rack ID where Voltage of the Rack with the highest number of strings which are under Partial Op due to limit of voltage difference alarm*)
	MesSystemCommandStatus		: WORD ; 		(* Command status*)
	MesSystemMode				: WORD;			(* (NA) bit0: ES caused by partial operation, bit1: ES caused by ES, bit2: ES caused by SPD, bit8: Status Ready, bit9: Status Idle, bit10: Staus Off-line*)
	MesSystemMode2				: WORD;			(* (NA) bit0: ES caused by partial operation, bit1: ES caused by ES, bit2: ES caused by SPD, bit8: Status Ready, bit9: Status Idle, bit10: Staus Off-line*)
	MesAlarm1					: WORD;			(* (NA) bit0:*)
	MesAlarm2					: WORD;			(* (NA) bit0:*)
	MesRackAlarm1				: WORD;			(* (NA) bit0:*)
	MesRackAlarm2				: WORD;			(* (NA) bit0:*)
	MesRackProtection1			: WORD;			(* (NA) bit0:*)
	MesRackProtection2			: WORD;			(* (NA) bit0:*)
	MesRackStringAlarm1			: WORD;			(* (NA) bit0:*)
	MesRackStringAlarm2			: WORD;			(* (NA) bit0:*)
	MesRackStringAlarm3			: WORD;			(* (NA) bit0:*)
	MesRackStringAlarm4			: WORD;			(* (NA) bit0:*)
	MesRackStringProtection1	: WORD;			(* (NA) bit0:*)
	MesRackStringProtection2	: WORD;			(* (NA) bit0:*)
	MesRackStringProtection3	: WORD;			(* (NA) bit0:*)
	MesRackStringProtection4	: WORD;			(* (NA) bit0:*)
	MesDiStatus					: WORD;			(* (NA) DI Status*)
	MesDoStatus					: WORD;			(* (NA) DI Status*)
	MesSystemConfig1			: WORD ; 		(* Samsung State word Config 1*)
	MesSystemConfig2			: WORD ;    	(* Samsung State word Config 2*)
	MesRackStringState			: WORD ;    	(* Samsung State word Rack state*)
	ParamNbRacks				: UINT ; 		(* Number of racks set in BBMS*)
	ParamNbModule				: UINT ; 		(* Number of modules per strings set in BBMS*)
	ParamStringNbMin			: UINT ; 		(* Minimal number of strings Operable in order to works set at BBMS*)
	ParamUdiff					: REAL ;		(* Maximum voltage difference between  string for connexion set in BBMS .*)
	
// Evaluate	
	MesUdcMin_RackID		: UINT:=1 ;			(* (NA) Id OF the Rack with the minimum Udc		// TO CALCULATE*)
	MesUdcMax_RackID		: UINT:=1 ;			(* (NA) Id of the Rack with the maximum Udc		// n'est pas ecrit*)
	CalEconnected 			: REAL ; 			(* Energy available for charge / discharge in the system BBMS.*)
	CalNbRackNormal			: UINT ; 			(* Number of racks without alarms .*)
	MesPdc					: REAL ; 			(*(kW) Cal : DC Power*)
	CalNbPointsDayCharge	: UINT;				(* {1 }(NA) Number of points per day of Charge*)
	CalNbPointsDayDischarge	: UINT;				(* {1 }(NA) Number of points per day of discharge*)
	CalNbPointsDayCenter	: UINT;				(* {1 }(NA) Number of points per day of Center*)
	CalNbPointsDayRest		: UINT;				(* {1 }(NA) Number of points per day of Rest*)
	CalCRateDischarge		: REAL;				(* {1 }daily average Discharge CRate*)
	CalCrateCharge			: REAL;				(* {1 }daily average Charge CRate*)
	CalRSoC					: REAL;				(* {1 }(%) daily average rest SoC*)
	CalCSoC					: REAL;				(* {1 }(%) daily average center SoC*)
	CalEnergyThroughput		: REAL;				(* {1 }(kWh) daily energy throughput*)
	

	
	AX_Rack					: ARRAY[1..CstNbRack_Pcs] OF RACK;	(* Object*)
	MesAlarmCode			: WORD;								(* (NA) Internal Akuo AlarmCode*)
	MesWarningCode			: WORD;								(* (NA) Internal Akuo WarningCode*)
	MesEventCode			: WORD;								(* (NA) Internal Akuo EventCode*)
	MesAlarmCom				: BOOL ;							(* Communication alarm*)
	MesCP_Read				: BOOL := FALSE;					(* Read function enable*)
	MesCP_Write				: BOOL := FALSE;					(* Write function enable*)
	
	
END_STRUCT
END_TYPE

// ---- 01_Equipement_Library/Datalogger/Datalogger.TcDUT
TYPE Datalogger :
STRUCT
	
	MesAlarmCode				: WORD ; 						(* Internal Akuo Alarm Code				*)
	MesWarningCode				: WORD ; 						(* Internal Akuo Warning Code       	*)
	MesEventCode				: WORD ; 						(* Internal Akuo Event Code         	*)
	 
	MesCP_Read					: BOOL; 						(* Permanent conditions for read		*)          

	MesCP_Write					: BOOL; 						(* Permanent conditions for read		*)    
                             						
END_STRUCT
END_TYPE

// ---- 01_Equipement_Library/Datalogger/Datalogger_PPCVerrerie.TcDUT
TYPE Datalogger_PPCVerrerie :
STRUCT
	MesData			: Datalogger ; 

	
	//225 kV 
//	PM_225kV									: PM ; // ION non remonté 
                                    			
	ProtectRelay_MainHVCB						: ProtectRelay_S42 ; 
	MainHVCB									: CB_MainHVCB_Sch ; 
                                    			
//	A1_GridHVCB									: GridHVCB ; Non remonté ? 
                                    			
	ProtectRelay_Transfo225kV					: ProtectRelay_T87 ; 
	Transfo_225kV								: Transfo_HV ; 	
	GRID										: GRID ; // non remonté ? 
	                                			
	                                			
                                    			
//	20 kV 		                    			
	MainMVCB									: MainMVCB_Sch ; 
	ProtectRelay_MainMVCB						: ProtectRelay_S42 ; 
						            			
	ProtectRelay_FeederMVCB						: ARRAY[1..2] OF ProtectRelay_S42 ; 		// 1. Midi 2. Plat 
	FeederMVCB									: ARRAY[1..2] OF FeederMVCB_Sch ; 
	                                	
                                    	
	                                	
	// Aux                          	
	Transfo_Aux									:  Transfo_MV ; 
	                                			
	UPS_CE										: UPS_VERR ; 
	UPS_TCM										: UPS_VERR ; 
	TapChanger 									: TapChanger ; 
	FSS											: FSS; 				(*Fire System*)
	DS											: TOR ; 			(*Door Sensor*)
	ES											: TOR ; 			(*Emergency Stop*)
	

	// Substation
	MesState									: WORD ; 			// Calculated  State of the HV + MV substation. 


	                                    		                   
	// 20 kV Courant Neutre et Cuve                                
    // transfo          ?????                                                    
	Mes20kVCourNeutCuveDefaultMasseCuve1		: BOOL;            	(*CourNeutCuveDefaultMasseCuve1	 	 *)
	Mes20kVCourNeutCuveMaxIexp2					: BOOL;            	(*CourNeutCuveMaxIexp2				 *)
	Mes20kVCourNeutCuveDefaultMasseCuve2		: BOOL;            	(*CourNeutCuveDefaultMasseCuve2	 	 *)
	Mes20kVCourNeutCuveMaxIexp4					: BOOL;            	(*CourNeutCuveMaxIexp4				 *)
	Mes20kVCourNeutCuveDefaultGround			: BOOL;            	(*CourNeutCuveDefaultGround		 	 *)
	Mes20kVCourNeutCuveMaxI0exp4				: BOOL;            	(*CourNeutCuveMaxI0exp4			 	 *)
	Mes20kVCourNeutCuveTempAlarm				: BOOL;            	(*CourNeutCuveTempAlarm			 	 *)
	Mes20kVCourNeutCuveTempTrigger				: BOOL;            	(*CourNeutCuveTempTrigger			 *)
	Mes20kVCourNeutCuveGazDischarge				: BOOL;            	(*CourNeutCuveGazDischarge			 *)
	Mes20kVCourNeutCuvePressure					: BOOL;   		   	(*CourNeutCuvePressure				 *)
	                                    		                   	
	Mes20kVCourNeutCuveI1						: REAL;            	(*(A) CourNeutCuveI1			 *)
	Mes20kVCourNeutCuveResidualI				: REAL;            	(*(A) CourNeutCuveResidualI	     *)
	Mes20kVCourNeutCuveDecltI1					: REAL;            	(*(A) CourNeutCuveDecltI1		 *)
	Mes20kVCourNeutCuveDecltI2					: REAL;            	(*(A) CourNeutCuveDecltI2		 *)
	                                                               	
	// Aux HT, BT and Transfo                                      	
	 // AuxMVCB                                                    	          
	MesAuxHTSect225kV							: BOOL;		       	(* AuxHTSect225kV						*)
	MesAuxHtSmaltHTBOpen						: BOOL;		       	(* AuxHtSmaltHTBOpen					*)
	MesAuxHtFusionFuseMeasures225kV				: BOOL;		       	(* AuxHtFusionFuseMeasures225kV			*)                                              
	MesAuxHtFusionFuseProtect225kV				: BOOL;		       	(* AuxHtFusionFuseProtect225kV			*)
	MesAuxHtFusionFuseCountRte225kV				: BOOL;		       	(* AuxHtFusionFuseCountRte225kV			*)
	MesAuxHtShortCircuitCurrentProtectCcp2		: BOOL;		       	(* AuxHtShortCircuitCurrentProtectCcp2	*)
	MesAuxHtDisjCount20kVOpen					: BOOL;		       	(* AuxHtDisjCount20kVOpen				*)
	MesAuxHtDisjRefVoltage20kVOpen				: BOOL;		       	(* AuxHtDisjRefVoltage20kVOpen			*)
	MesAuxHtShortCircuitCurrentProtectCcp3		: BOOL;		       	(* AuxHtShortCircuitCurrentProtectCcp3	*)
                                                                   	
	MesAuxBtTriggerGeneralDisj					: BOOL;		       	(*AuxBtTriggerGeneralDisj				 *)
	MesAuxBt400VManqueAC						: BOOL;		       	(*AuxBt400VManqueAC					     *)
	MesAuxBt400VDecltAntenneScada				: BOOL;		       	(*AuxBt400VDecltAntenneScada			 *)
	MesAuxBt400VDecltAntennePrio				: BOOL;		       	(*AuxBt400VDecltAntennePrio			 	 *)
	MesAuxBt400VPermutAutoStopMode				: BOOL;		       	(*AuxBt400VPermutAutoStopMode			 *)
	MesAuxBt400VPermutAutoNormalMode			: BOOL;		       	(*AuxBt400VPermutAutoNormalMode		 	 *)
	MesAuxBt400VPermutAutoSecoursMode			: BOOL;		       	(*AuxBt400VPermutAutoSecoursMode		 *)
	MesAuxBt400VPermutModeAuto					: BOOL;    	       	(*AuxBt400VPermutModeAuto				 *)
	MesAuxBt400VVoltageLossNormalAlim			: BOOL;		       	(*AuxBt400VVoltageLossNormalAlim		 *)
	MesAuxBt400VVoltageLossSecoursAlim			: BOOL;		       	(*AuxBt400VVoltageLossSecoursAlim		 *)
	MesAuxBt400VDefaultPermut					: BOOL;		       	(*AuxBt400VDefaultPermut				 *)


	MesAuxBtDefaultInverter						: BOOL;  		   	(* AuxBtDefaultInverter	*)
                                                                   	
	MesAuxBtSyntDefaultDistrib48VccJdb			: BOOL;  		   	(* AuxBtSyntDefaultDistrib48VccJdb		*)
	MesAuxBtSyntOpenDistrib48VccJdb				: BOOL;		       	(* AuxBtSyntOpenDistrib48VccJdb			*)
	MesAuxBtSyntDefaultDistrib48VccLocker		: BOOL;  		   	(* AuxBtSyntDefaultDistrib48VccLocker	*)
    MesAuxBtSyntOpenDistrib48VccLocker			: BOOL;		       	(* AuxBtSyntOpenDistrib48VccLocker		*)
                                                                   	
	MesAuxTransfoMeltingFusesContact			: BOOL;		       	(* AuxTransfoMeltingFusesContact	*)
                                                                   	
	MesAuxTransfoSwitchGear						: BOOL;	           	(*AuxTransfoSwitchGear		 *)
                                                                   	
	MesAuxHtOpenSectLine225kV					: BOOL;		       	(* AuxHtOpenSectLine225kV*)
	MesAuxHtCloseSectLine225kV					: BOOL;		       	(* AuxHtCloseSectLine225kV*)
                                                                   	
	                                                               	
	MesAuxHtOpenSectMalt						: BOOL;		       	(* AuxHtOpenSectMalt*)
	MesAuxHtCloseSectMalt						: BOOL;		       	(* AuxHtCloseSectMalt*)
                                                                   	
	MesAuxHtTeleCondamnSl225kV				 	: BOOL;		       	(* AuxHtTeleCondamnSl225kV			*)
	MesAuxHtDeTeleCondamnSl225kV				: BOOL;            	(* AuxHtDeTeleCondamnSl225kV		*)
	MesAuxHtTelecommandeRelestActif				: BOOL;		       	(* AuxHtTelecommandeRelestActif		*)
	MesAuxHtTelecommandeRelestPassif			: BOOL;	           	(* AuxHtTelecommandeRelestPassif	*)
	                                                               
	// Door Sensor, Fire Alarm, Local/Remote, Emergency Stop	   
	                                                            
	MesLocalRemoteOperation                  	: BOOL;            	(*LocalRemoteOperation    *)


	MesAlarmCom									: BOOL ; 		   	(* Communication Error with I35 module *) 
	MesCP_Read									: BOOL ;  			(* Cal : Read function enable *)

	MesAlarmCode1								: WORD ; 			(* Internal Akuo Alarm Code   *)
	MesAlarmCode2								: WORD ; 			(* Internal Akuo Alarm Code   *)
	MesAlarmCode3								: WORD ; 			(* Internal Akuo Alarm Code   *)
	MesWarningCode1								: WORD ; 			(* Internal Akuo Warning Code *)
	MesWarningCode2								: WORD ; 			(* Internal Akuo Warning Code *)  
	MesWarningCode3								: WORD ; 			(* Internal Akuo Warning Code *)
	MesWarningCode4								: WORD ; 			(* Internal Akuo Warning Code *)  
	MesWarningCode5								: WORD ; 			(* Internal Akuo Warning Code *) 
    MesWarningCode6								: WORD ; 			(* Internal Akuo Warning Code *)     
	MesEventCode1								: WORD ; 			(* Internal Akuo Event Code   *)  
	MesEventCode2								: WORD ; 			(* Internal Akuo Event Code   *) 
	MesEventCode3								: WORD ; 			(* Internal Akuo Event Code   *)  			                                                   			                                               
	
END_STRUCT
END_TYPE

// ---- 01_Equipement_Library/Datalogger/Datalogger_SchSkid.TcDUT
TYPE Datalogger_SchSkid :
STRUCT

	MesData							: Datalogger ; 							(* MesData *)
                        			                			
	MesComutLocal					: BOOL; 								(* FALSE := Local, TRUE := Remote (DI_204) *)
	MesState_MVCB					: BOOL; 								(* True := Fermé, False := Ouvert (DI_205) *)
	MesWatchdog_ProtectRelayVIP		: BOOL; 								(* WatchDog of VIP410 (DI_201)			   *)
	MesFault_ProtectRelayVIP		: BOOL; 								(* TRUE:= Fault, False:= OK, Déclenchement du défaut VIP (DI_206) *)
	                        			
	MesToggleRead					: BOOL; 								(* Cal State com of FB IO *)
	MesToggleWrite					: BOOL;;  								(* Cal State com of FB IO *)
	 
	DS_Synthesis					: TOR ; 								(* Synthesis of door sensors True = a door is opened (DI_209) 			 *)
	CB_INV							: ARRAY[1..CstNbInv_PTR_G] OF  TOR; 	(* TRUE := CB opened, False : CB closed, INV 1 (DI_202) / INV 2 (DI_203) *)
	Transfo_Synthesis				: Transfo_MV; 							(* Transfo *)
	 	 						
END_STRUCT
END_TYPE

// ---- 01_Equipement_Library/Datalogger/Datalogger_SENECA.TcDUT
TYPE Datalogger_SENECA :
STRUCT
	
	MesData			: Datalogger ; 			  (* (NA) MesData *)
                        			                			                            	
	MesWindSp		: REAL ;				  (* (km/h) Wind speed of the weather station on SPP zone	 		*)
	MesWindDir		: REAL ;  				  (* (deg) Wind direction of the weather station on SPP zone	    *)
	 	 						
END_STRUCT
END_TYPE

// ---- 01_Equipement_Library/Fan/Fan.TcDUT
TYPE Fan :
STRUCT
		MesIsRun			: BOOL ;	(* Fan is running status*)
		MesTemp				: REAL ; 	(*(°C) Temperature // fTmp_Max*)
        MesStartTime 		: WORD ;	(* Cal: Starting Time*)
        MesStopTime 		: WORD ;	(* Cal : Stopping Time*)
		
		MesAlarmCode		: WORD ;    (* (NA) Internal Akuo AlarmCode*)
		MesWarningCode		: WORD ;    (* (NA) Internal Akuo WarningCode*)
		MesEventCode		: WORD ;    (* (NA) Internal Akuo EventCode*)
		
		
END_STRUCT
END_TYPE

// ---- 01_Equipement_Library/GRID/GRID.TcDUT
///////////
// Structure For DEIECommand. Main Operating Data to be saved (ex: OPC)  
//////////
TYPE GRID :
STRUCT
	// TC
	OUT_CmdAutCpl			 	: BOOL ;			(* (NA) Autorisation couplage (pulse)*)
	OUT_CmdDisconnect		 	: BOOL ;			(* (NA) Disconnect command (pulse)*)
	OUT_CmdEmergencyDisconnect	: BOOL ;			(* (NA) Emergency disconnect command (pulse)*)	
	OUT_SetptP 				 	: REAL ;			(* (kW) P Setpoint from EDF*)
	OUT_SetptQ 				 	: REAL ;			(* (kVar) Q Setpoint from EDF*)
	OUT_MesPPUnavailable		: BOOL ;			(* (NA) TS centrale indisponible*)
	OUT_MesPPConnected			: BOOL ; 			(* (NA)Centrale couplée(1)/Centrale Découplée(0)*)	
	
	// State 	
	MesAlarmCode				: WORD ; 			(* (NA) Internal Akuo Alarm Code*)
	MesWarningCode 			 	: WORD ; 			(* (NA) Internal Akuo Warning Code*)
	MesEventCode			 	: WORD ;			(* (NA) Internal Akuo Warning Code*)
	MesEventCode2				: WORD ; 			(* (NA) EventCode 2*)

	MesAlarmCom				 	: BOOL ;			(* (NA) Communication alarm *)
	MesCP_Read				 	: BOOL := TRUE; 	(* (NA) Cal : Read function enable*)
	
END_STRUCT
END_TYPE

// ---- 01_Equipement_Library/GRID/GRID_Enedis.TcDUT
///////////
// Structure For DEIECommand. Main Operating Data to be saved (ex: OPC).
//////////
TYPE GRID_Enedis :
STRUCT
	
	MesData								: GRID ; 		(* GRID MesData *)
                                       	
	OUT_CmdPReg                         : BOOL ;     	(* (NA) Passage à P0 reçu DI*)
	OUT_CmdQReg	                   	    : BOOL ;     	(* (NA) Passage à Q0 reçu DI*)

	OUT_Rse								: BOOL; 		(* (NA) Protection en Rse(1) / Protection Hors RSE (O) *)
	OUT_TA								: BOOL; 		(* (NA) Telecaction en service (1) / Teleaction Hors service (0)*)
	
END_STRUCT
END_TYPE

// ---- 01_Equipement_Library/HVAC/HVAC.TcDUT
TYPE HVAC :
STRUCT

	MesSetptTemp		: REAL ;    	 (*(°C)  Temperature setpoint*)

	MesSetptHygro		: REAL ;    	 (*(%)   Hygrometry setpoint      *)

	MesOn				: BOOL ;    	 (*      HVAC is on *)

	MesAlarmCom			: BOOL ;    	 (*      Communication alarm *)

	WorkingHr 			: TIME ; 		 (* 	 Time AC has been on*)
	MesCP_Read			: BOOL := FALSE; (* 	 Read function enable*)
	MesCP_Write			: BOOL := FALSE; (* 	 Write function enable*)
	
	MesAlarmCode		: WORD ;		 (* 	 AlarmCode for the TGBT*)
	MesWarningCode		: WORD ;		 (* 	 WarningCode for the TGBT*)
	                                     

	
END_STRUCT
END_TYPE

// ---- 01_Equipement_Library/HVAC/HVAC_MADI.TcDUT
TYPE HVAC_MADI :
STRUCT
	MesData				: HVAC ;	

	MesHygro_Amb		: REAL ; 		 (*(%)	 Hygro value*)
	MesPressure1		: REAL ; 		 (*(bar) Pressure of the evaporatr 1 (bar )*)
	MesTemp_Room		: REAL ; 		 (*(°C)	 Temperature value .*)
	MesTemp_Outlet		: REAL ; 		 (*(°C)  Temperature at the HVAC output*)
	MesTemp_Outside		: REAL ; 		 (*(°C)  Outside air temperature*)
	
	MesSetptTempmin		: REAL ;    	 (*(°C)  Min Temperature setpoint *)
	MesSetptTempmax		: REAL ;    	 (*(°C)	 Max Temperature setpoint *)
	
	MesSetptHygromin	: REAL ;    	 (*(%)	 Min Hygrometry setpoint  *)
	MesSetptHygromax	: REAL ;    	 (*(%)	 Max Hygrometry setpoint  *)
	
	MesAlarmsSynthesis	: BOOL ;         (*      Alamrs synthesis *)
	
	MesCooling			: BOOL ;   		 (*()	 The HVAC is cooling the air*)
	MesHeating			: BOOL ; 		 (*()	 The HVAC is heating the air*)
	                                     
	MesAlarm1			: WORD ; 		 (* 	 HVAC Alarm word 1*)
	MesAlarm2			: WORD ; 		 (* 	 HVAC Alarm word 2*)
	MesAlarm3			: WORD ; 		 (* 	 HVAC Alarm word 3*)
	
END_STRUCT
END_TYPE

// ---- 01_Equipement_Library/HVAC/HVAC_Standard.TcDUT
TYPE HVAC_Standard :
STRUCT
	MesData				: HVAC ;	

	MesHygro_Amb		: REAL ; 		 (*(%)	 Hygro value*)
	MesPressure1		: REAL ; 		 (*(bar) Pressure of the evaporatr 1 (bar )*)
	MesTemp_Room		: REAL ; 		 (*(°C)	 Temperature value .*)
	MesTemp_Outlet		: REAL ; 		 (*(°C)  Temperature at the HVAC output*)
	MesTemp_Outside		: REAL ; 		 (*(°C)  Outside air temperature*)
	
	MesSetptTempmin		: REAL ;    	 (*(°C)  Min Temperature setpoint *)
	MesSetptTempmax		: REAL ;    	 (*(°C)	 Max Temperature setpoint *)
	
	MesSetptHygromin	: REAL ;    	 (*(%)	 Min Hygrometry setpoint  *)
	MesSetptHygromax	: REAL ;    	 (*(%)	 Max Hygrometry setpoint  *)
	
	MesAlarmsSynthesis	: BOOL ;         (*      Alamrs synthesis *)
	
	MesCooling			: BOOL ;   		 (*()	 The HVAC is cooling the air*)
	MesHeating			: BOOL ; 		 (*()	 The HVAC is heating the air*)
	                                     
	MesAlarm1			: WORD ; 		 (* 	 HVAC Alarm word 1*)
	MesAlarm2			: WORD ; 		 (* 	 HVAC Alarm word 2*)
	MesAlarm3			: WORD ; 		 (* 	 HVAC Alarm word 3*)
	
END_STRUCT
END_TYPE

// ---- 01_Equipement_Library/Inverter/INV.TcDUT
///////////
// Structure For Inverter. Main Operating Data to be saved (ex: OPC).  
//////////
TYPE INV :
STRUCT
	
		// INV Measures from Datalogger
		MesP 				: REAL ; 		(* (kW) 	Active Power output (AC) of inverter PCS01*)
		MesQ 				: REAL ;  		(* (kVAr)   Reactive AC Power Produced				  *)
		MesPdc 				: REAL ;  		(* (kW) 	Power measure (DC) of inverter			  *)
		MesIdc 				: REAL ;	 	(* (A) 	    Total Current measure (DC)				  *)
		MesUdc 				: REAL ;  		(* (V)  	Mean Voltage measure (DC)				  *)
		MesU 				: REAL ;		(* (V) 	    Mean Voltage measure (AC)				  *)
		MesV				: REAL ; 		(* (V)      Mean Phase to Neutral voltage			  *)
		MesI				: REAL ;		(* (A)      Mean Phase Current						  *)
		MesI0               : REAL ;        (* (A) 		Residual current						  *) 
		MesFreq				: REAL ; 		(* (Hz)     Frequency                                 *)
		MesS				: REAL ; 		(* (kVA)     Apparent Power						      *)
		MesInsuResistor		: REAL ; 		(* (MOhms) Insulation Resistance					  *)
		MesCosPhi			: REAL ; 		(* (p.u) Power Factor								  *)
		MesTemp				: REAL ; 		(* (C) Inverter Temperature							  *)
		MesState			: UINT ;		(* (NA) Inverter Status								  *)
		ParamPn				: REAL ; 		(* (kW) Nominal Capacity of SMA 25000 TL Inverter	  *)
		ParamQn				: REAL ;		(* (kVAr) Nominal reactive power 					  *)
		MesCurtl		    : BOOL ; 		(* (NA)Cal True if the inverter is curtailing Power	  *)
		MesAlarmCom			: BOOL ; 		(* (NA) Communication Alarm							  *)
		MesCP_Read			: BOOL := TRUE;	(* (NA) Cal : Permanent Condition for Read			  *)
		MesCP_Write			: BOOL := TRUE;	(* (NA) Cal : Permanenent Condition for Write		  *)
		                                                                                        
		MesOpened_Ac        : BOOL ;   		(* (NA) Ac switch is opened							  *)
		MesOpened_Dc        : BOOL ;   		(* (NA) Dc switch is opened							  *)
		                                                                                        
		OUT_CmdStart        : BOOL ;        (* (NA) OUT start command 							  *)
		OUT_CmdStop         : BOOL ;        (* (NA) OUT stop command   							  *)
		OUT_SetptP    	    : REAL ;        (* (kW) OUT P setpoint  							  *)
		OUT_SetptQ          : REAL ;        (* (kVAr)  OUT Q setpoint   						  *)
		//MesState			: UINT ; 		(* (NA) Cal: Akuo Internal State . O=Stopped, 1 = RUN *)
		MesAlarmCode		: WORD ; 		(* (NA) Internal Akuo AlarmCode                       *)
		MesWarningCode		: WORD ; 		(* (NA) Internal Akuo WarningCode                     *)
		MesEventCode		: WORD ; 		(* (NA) Internal Akuo EventCode                       *)

END_STRUCT
END_TYPE

// ---- 01_Equipement_Library/Inverter/INV_1000CP_XT.TcDUT
TYPE INV_1000CP_XT :
	//SMA CP, CP-US, CP-JP and HE-20
STRUCT
		Mesdata					: INV;
		BJMonitor				: INV_1000CP_XT_StringMonitor;	

// Device Family
		MesEventID				: REAL;		(* Event ID of the current event [ErrNo]*)
		MesWaitGridTm			: TIME; 	(* Time until grid connection attempt (s) [TmsRmg].*)
	// Setpoint ??? RecoAction
		SetptRecoAction			: REAL;		(* 336 = Contact the manufacturer,337 = Contact the installer,338 = Invalid [Prio]*)
		MesOpened_CBGrid		: BOOL;     (* 51 = Contactor closed,311 = Contactor open [GriSwStt]*)
		MesRiso					: REAL;		(* Insulation resistance (Ohm) [Riso]*)
		MesState_KeyComut		: BOOL;     (* Status of key switch :381 = Stop,569 = Activated [DInKeySwStrStp]*)
		MesState_Inv			: REAL;		(* Operating state, 309 = Operation,381 = Stop,455 = Warning,1392 = Error,1393 = Wait for PV voltage,1394 = Wait for AC grid,1480 = "Wait for electricity supplier" operating state (for 0% regulation),1560 = Remote shutdown active,2383 = Manual restart [mode]*)
		MesIDError				: REAL;     (* Error location OF the present error,267 = Inverter , 1395 = DC section,1396 = AC grid [Error]*)
		MesEventID_INVSMA		: REAL;		(* Current, complete event number [ErrNoSma]*)
		MesOpened_GFDI			: BOOL;     (* Switching status of the GFDI  (311: Open & 51 : Close) [DInGfdi]*)
		MesOpened_CBdc			: BOOL;		(* DC Switch status (51: Close, 311: Open) [DcSwStt]*)
		MesState_Restart		: REAL;		(* Status of current restart interlock :1690 = Fast shut-down, 2386 = Overvoltage, 2387 = Undervoltage, 2388 = Overfrequency, 2389 = Underfrequency, 2390 = Passive islanding detection, 2490 = Phase lost detection [ManResStt]*)
		MesOpened_CBac			: BOOL;  	(* AC switch-disconnector in cabinet [AcDiscon]: 51 = Closed, 311 = Open*)
		MesEActTot				: REAL;     (* Total yield (MWh) [E-Total]*)
		MesEActDay				: REAL;     (* Daily yield (Wh) [E-heute]*)
		MesWorkingHr			: TIME;     (* Operating time (Hr) [h-On]*)
		MesFeedTm				: TIME;     (* Feed-in Time (Hr) []*)
		MesWorkingHr_Fan1		: TIME;     (* Operating time of the interior fan 1 (Hr) [CntFanCab1]*)
		MesWorkingHr_Fan2		: TIME;     (* Operating time of the interior fan 2 (Hr) [CntFanCab2]*)
		MesWorkingHr_Heat		: TIME;		(* Operating time of the interior heater (Hr) [CntFanHs]*)
		MesWorkingHr_Heat2		: TIME;		(* Operating time of the interior heater (Hr) [CntHtCab2]*)
		MesWorkingHr_Fan3		: TIME;     (* Operating time of interior fan 3 (h) [CntFanCab3]*)
		MesIdc					: REAL;		(* (A) DC Current [Ipv]*)
		MesUdc					: REAL;		(* (V) DC Voltage [Vpv]*)
		MesPdc					: REAL;		(* (kW) DC Power [Ppv]*)
		MesP					: REAL;		(* (kW) AC POWER*)
		MesQ					: REAL;		(* (kvar) AC Reactive power*)
		MesU12					: REAL;     (* (V) Line to line Voltage L1-L2 utility grid VacL12*)
		MesU23					: REAL;     (* (V) Line to line Voltage L2-L3 utility grid VacL23*)
		MesU31					: REAL;     (* (V) Line to line Voltage L3-L1 utility grid VacL31*)
		MesV					: REAL;		(* (V) AC Voltages of each line*)
		MesI					: REAL;		(* (A) Line current [Iac]*)
		MesI1					: REAL;		(* (A) Mean AC current L1 Total [IacL1]*)
		MesI2					: REAL;		(* (A) Mean AC current L2 Total [IacL2]*)
		MesI3					: REAL;		(* (A) Mean AC current L3 Total [IacL3]*)
		MesFreq					: REAL;		(* (Hz) Power frequency [Fac]*)
		MesCosPhi				: REAL;     (* (NA) Power factor	[PF]*)
		MesTypeCosPhi			: REAL;		(* Setpoint excitation type of cos φ [PF-PFExtSpt]: 1041 = Capacative, 1042 = Inductive*)
		MesQMode	           	: REAL;		(* Operating mode of the reactive power regulation [Q-VArMod]:303 = Off,1069= Reactive power-/voltage characteristic curve Q(V),1070 = Reactive power Q, direct setpoint,1071 = Reactive power const. Q (kVAr)                                                          *)
											(* 1072 = Reactive power Q, setpoint via system control, 1074 = cos φ, direct setpoint, 1075 = cos φ, setpoint via system control, 1076 = cos φ(P) – characteristic curve, 1387 = Reactive power Q, setpoint via analog input , 1388 =cos φ, setpoint via analog input, *)
											(* 1389 = Reactive power-/voltage characteristic curve Q(V) with hysteresis and deadband*)
		MesSetptQ				: REAL;     (* Reactive power setpoint (kVAr) [SpntPwrRt]*)
		MesSetptQ_Pct			: REAL;     (* Reactive power setpoint (%) [Q-VArNom].*)
		MesSetptCosPhi			: REAL;		(* Setpoint cos φ [PF-PFSpt]*)
		MesSetptType_CosPhi		: REAL;		(* Setpoint excitation type of cos φ [PF-PFExtSpt]: 1041 = Capacative, 1042 = Inductive*)
		MesPMode				: REAL;		(*	 [P-WMod]: 303 = Off, 1077 = Active power limitation P (kW), 1078 = Active power limitation P in (%) of PMAX,*)
											(*	1079 = Active power limitation P via plant control, 1390 = Active power limitation P via analog input*)

// Stopped here											(*	1391 = Active power limitation P via digital inputs*)
		MesPSetpt				: REAL;     (* (kW) Active power setpoint [P-WSp]*)
		MesPSetptPct			: REAL;     (* (%) Active power setpoint  [P-WNom].*)
		MesTmpHs				: REAL;		(* (°C) Heat sink temperature 1 [TmpHs]*)
		MesTmpCab1				: REAL;		(* (°C) Heat sink temperature Cab 1 [TmpCab1]*)
		MesTmpCab3				: REAL;		(* (°C) Heat sink temperature Cab 3 [TmpCab3]*)
		MesTmpExt				: REAL;		(* (°C) External temperature 1 [TmpExt1]*)
		MesTmpCol				: REAL;		(* (°C) Temperautre of the sinusoidal filter choke [TmpCol]*)
		MesGHI					: REAL;		(* (W/m²) Total irradiation of the sensor surface [ExtSolIrr]*)
		MesInCur1				: REAL;		(* (mA) Analog current Input 1 [ExtSolIrr]*)
		MesInCur2				: REAL;		(* (mA) Analog current Input 2 [ExLAnaInCur]*)
		MesOpStateOn			: BOOL;		(* (NA) Operating state : 381 = Stop,569 = Activated  [SpntRemEna]*)
		MesbRIsoOn				: BOOL;		(* (NA) External measurement of the insulation resistance : 303=Off, 308=On*)
		//AX_BJ					: ARRAY [1..8] OF REAL; // (A) Current of each BJ*)

		
END_STRUCT
END_TYPE

// ---- 01_Equipement_Library/Inverter/INV_1000CP_XT_StringMonitor.TcDUT
TYPE INV_1000CP_XT_StringMonitor:
STRUCT
	STR : ARRAY [1..9] OF STR;
	MesAlarmContact_1			: BOOL; (*303 = Off, 308 = On*)
	MesAlarmContact_2			: BOOL; (*303 = Off, 308 = On*)
END_STRUCT
END_TYPE

// ---- 01_Equipement_Library/Inverter/INV_Huawei.TcDUT
///////////
// Structure For Inverter. Main Operating Data to be saved ( ex: OPC ) .  
//////////
TYPE INV_Huawei :
STRUCT
	
	// INV Measures
		MesData			: INV ; (* INV *) 

		STR				: ARRAY[1..12 ] OF STR ;  	(* STR *) 
		
		MesEDay			: REAL ;	    			(* (kWh)Daily Energy	*)
	    MesETot			: REAL ;					(* (kWh)Total Energy	*)
		MesI1			: REAL ;					(*	(A) MesI1			*)
		MesI2			: REAL ;					(*	(A) MesI2			*)
	    MesI3			: REAL ;					(*	(A) MesI3			*)
		MesU12			: REAL ;					(*	(V) MesU12			*)
        MesU23			: REAL ;					(*	(V) MesU23			*)
        MesU31			: REAL ;					(*	(V) MesU31			*)
		MesV1			: REAL ;					(*	(V) MesV1			*)
		MesV2			: REAL ;					(*	(V) MesV2			*)
		MesV3			: REAL ;					(*	(V) MesV3			*)
                                        			
		MesStateIndic 	: WORD ;					(*	MesStateIndic 		*)
		MesOpeStatus 	: WORD ;					(*	MesOpeStatus 		*)
		MesAlm1			: WORD ;					(*	MesAlm1				*)
		MesAlm2			: WORD ;					(*	MesAlm2				*)
		MesAlm3			: WORD ;					(*	MesAlm3				*)
	                                                        	
		
		
	
		
		
		


END_STRUCT
END_TYPE

// ---- 01_Equipement_Library/Inverter/INV_Sch4400.TcDUT
///////////
// Structure For Inverter. Main Operating Data to be saved (ex: OPC).  
//////////
TYPE INV_Sch4400 :
STRUCT
	
	// INV Measures
	MesData					: INV ;					(* MesData *) 
		            		
	STR						: ARRAY[1..10] OF STR;	(* (NA) Strings *)

	//Electrical Measurements
	MesI1					: REAL; (* (A) Phase A RMS current at inverter side of AC circuit breaker CB501								*)
	MesI2					: REAL; (* (A) Phase B RMS current at inverter side of AC circuit breaker CB501                             *)
	MesI3					: REAL; (* (A) Phase C RMS current at inverter side of AC circuit breaker CB501                             *)
	MesV1					: REAL; (* (V) Phase A RMSvoltage (line to virtual neutral)at grid side of AC circuit breaker CB501         *)
	MesV2					: REAL; (* (V) Phase B RMSvoltage (line to virtual neutral)at grid side of AC circuit breaker CB501         *)
	MesV3					: REAL; (* (V) Phase C RMSvoltage (line to virtual neutral)at grid side of AC circuit breaker CB501         *)
	MesU12					: REAL; (* (V) Phase AB RMS voltage (line to line)at grid side of AC circuit breaker CB501                  *)
	MesU23					: REAL; (* (V) Phase BC RMS voltage (line to line)at grid side of AC circuit breaker CB501                  *)
	MesU31					: REAL; (* (V) Phase CA RMS voltage (line to line)at grid side of AC circuit breaker CB501                  *)
	
	//Production Measurements
	MesEActProd				: REAL; (* (Wh) Active energy delivered.Integrates positive values of GenMMTR/DmdWhFil.Ignores negative values		*)
	MesEActCons				: REAL; (* (Wh) Active energy consumed.Integrates negative values of GenMMTR/DmdWhFil.Ignores positive values       *)
	MesEReactProd			: REAL; (* (VArh) Reactive energy delivered.Integrates positive values of GenMMTR/DmdVAhFil.Ignores negative values *)
	MesEReactCons			: REAL; (* (VArh) Reactive energy consumed.Integratesnegative values of GenMMTR/DmdVAhFil.Ignores positive values   *)
	MesEday					: REAL; (* (Wh) Active energy produced during the day                                                               *)
	
	//Communication Status
	MesStateCom				: BOOL; (* (NA) False := Not communicating, True := Communicating 	*)
	
	//Status Summary
	MesStateCBac			: BOOL; (* (NA) False := Open; True := Close, Status of event139 "CB501 Closed". AC circuit breaker CB501 is closed /INVx/AcXCBR/ClsActVal				 *)
	MesStateCBdc			: BOOL; (* (NA) False := Open; True := Close, Status of event140 "CB201 Closed". DC circuit breaker CB201 is closed /INVx/DcXCBR/ClsActVal               *)
	MesEarthing_Relay		: BOOL; (* (NA) False := Open; True := Close, Status of event157 "K202 Closed". Ground relay K202 is closed /INVx/GndXSWI/ClsActVal                      *)
	MesFaultGnd				: BOOL; (* (NA) False := Alert; True := No alert, Ground fault status. Digital outputDO_121 follows the state of this register /INVx/RcdMMXU/GndFltDrvSt *)
	MesStateNoAlert			: BOOL; (* (NA) False := Alert iverter has detected an abnormal event which prevents operation. ; True := No alert. /INVx/GenGGIO/NoFltDrvSt             *)
	MesState				: UINT; (* (NA) This parameter should be used for informational status only //INVx/GenZINV/Stt                                                           *)
	MesBdrigeCtlMod			: UINT;	(* (NA) Inverter bridge control mode /INVx/GenZINV/CtlMod                                                                                        *)
	MesWorkingHr			: REAL; (* (Hr) Total duration that the inverter has been online since power up /INVx/GenGAPC/TmsCnt                                                	 *)
	MesEvendID				: REAL;	(* (NA) Event ID of the currently active event. /INVx/EvtGGIO/ActId                                                                              *)
	MesEventID_Stop			: REAL;	(* (NA) Event ID of the first event that caused the Inv to go offline (normal or not)/INVx/EvtGGIO/OflStrActId                                   *)
	MesStateID_Recovery		: REAL;	(* (NA) Procedure for the Inv to recover: 0:No stop event, 1:Automatic, 2:Manual (=acknowledge), 3:Local (= physique) /INVx/EvtGGIO/RecovActTyp  *)
	MesEventID_AbnormalOff	: REAL;	(* (NA) Abnormal offline status ID: ID of the event that caused an abnormal stop (0=No abnormal stop) /INVx/EvtGGIO/OflForcSt                    *)
	MesState_TypeSetptP		: REAL;	(* (NA) Dominant limit or setpoint affecting active power production : 0: None, 11: CmdSetpt from comm, 15: MPPT /INVx/WMMXU/PriConId            *)
	MesSetptP				: REAL;	(* (pu) Value of the dominant active power limit W                                                                                    			 *)
	MesState_TypeSetptQ		: REAL; (* (NA) Dominant limit or setpoint affecting reactive power production : 0: None, 6: CmdSetpt from comm                                     	 *)
	MesSetptQ				: REAL;	(* (pu) Value of the dominant reactive power limit VAr                                                                                			 *)
	
	MesStartDisabled		: BOOL; (* (NA) Start disable : False := Start can be abled 						 *)
	MesStartDisabledPersis	: BOOL; (* (NA) Persistent start disable : must be the same as MesStartDisabled      *)
	
	// System Commands
	// Persistent value of inverter enable command.The value set here defines the initial value of GenZINV/Ena when the inverter powers on
	MesSetptP_CC 			: REAL;			(* (kW)   value of active power COMMAND																 *)
	MesSetptQ_CC 			: REAL;			(* (kVar) value of reactive power COMMAND                                                            *)
	MesSetptCosPhi_CC 		: REAL; 		(* (NA)  Power factor                                                            					 *)
	ParamID_QType			: UINT := 1; 	(* (NA) reactive power is defined by : 1: Q command mode, 2: PF command mode, 3: Q(P) command mode   *)
	ParamTP_RampP			: REAL; 		(* (s) Duration for the active power to reach the new setpoint                 						 *)
	ParamTP_RampCosPhi		: REAL; 		(* (s) Duration for the active power to reach the new setpoint                 						 *)
	ParamTP_RampQ			: REAL; 		(* (s) Duration for the active power to reach the new setpoint                 						 *)
	                		        		
	//Temp          		        		
	MesTempExt				: REAL;			(* (C°) External temperature *)
			
END_STRUCT
END_TYPE

// ---- 01_Equipement_Library/Inverter/SL_Huawei.TcDUT
///////////
// Structure For Inverter. Main Operating Data to be saved ( ex: OPC ) .  
//////////
TYPE SL_Huawei :
STRUCT
	
		MesData				: INV ;  (* INV *) 
	
	// INV Measures
		MesEDay				: REAL ;     	(*/ (kWh) Daily Energy*)
	    MesETot				: REAL ;		(*/ (kWh) Total Energy*)
		MesOn				: BOOL ;        (* Smartlogger is ON*)
		MesI1				: REAL ;        (* (A) AC current phase 1*)
		MesI2				: REAL ;        (* (A) AC current phase 1*)
	    MesI3				: REAL ;        (* (A) AC current phase 1*)
		MesU12				: REAL ;        (*(V) AC Voltage phase1 to phase2*)
        MesU23				: REAL ;        (*(V) AC Voltage phase2 to phase3*)
        MesU31				: REAL ;        (*(V) AC Voltage phase3 to phase1*)
		MesEff				: REAL ; 		(* (%) Inverter efficiency*)
		MesSetptPMax		: REAL ;        (* (kW) Maximal Active power setpoint*)
		MesSetptQMax		: REAL ;        (*(kVAr) Maximal reactive power setpoint*)
		MesSetptQMin		: REAL ;        (*(kVAr) Minimal reactive power setpoint*)
		OUT_SetptPlimit		: REAL ;        (*(kW) Maximal Active power setpoint sent by PPC*)
		OUT_SetptQlimit		: REAL ;        (*(kVAr) Maximal Reactive power setpoint sent by PPC*)

END_STRUCT
END_TYPE

// ---- 01_Equipement_Library/Inverter/STR.TcDUT
TYPE STR :
STRUCT
		MesIdc			: REAL;   						(* (A) DC current *)
		MesUdc			: REAL;							(* (V) DC voltage *)
END_STRUCT
END_TYPE

// ---- 01_Equipement_Library/IPC/IPC.TcDUT
TYPE IPC :
STRUCT
		
		MesAlarmCode		: WORD ;	(* (NA) Internal Akuo AlarmCode		*)
		MesWarningCode		: WORD ; 	(* (NA) Internal Akuo WarningCode   *)
		MesEventCode		: WORD ; 	(* (NA) Internal Akuo EventCode	    *)
		
END_STRUCT
END_TYPE

// ---- 01_Equipement_Library/Operation Meter/PM.TcDUT
///////////
// Structure For I35. Main Operating Data to be saved (ex: OPC).  
//////////
TYPE PM :
STRUCT
		MesU12						: REAL ; (* (V) Phase1 - Phase 2 AC Voltage 		   			*)
		MesU23						: REAL ; (* (V) Phase2 - Phase 3 AC Voltage         			*)
		MesU31						: REAL ; (* (V) Phase3 - Phase 1 AC Voltage         			*)
  		MesV1						: REAL ; (* (V) Phase1 AC Voltage                   			*)
		MesV2						: REAL ; (* (V) Phase2 AC Voltage                   			*)
		MesV3						: REAL ; (* (V) Phase3 AC Voltage		           				*)
		MesFreq						: REAL ; (* (Hz)Frequency		                   				*)
		MesI1						: REAL ; (* (A) AC current Phase 1                  			*)
		MesI2						: REAL ; (* (A) AC current Phase 2                  			*)
		MesI3						: REAL ; (* (A) AC current Phase 3                  			*)
		MesIn						: REAL ; (* (A) Neutral AC current                  			*)
		MesP						: REAL ; (* (kW) Total Active power                 			*)
		MesQ						: REAL ; (* (kVAr) Total Reactive Power Phase 1     			*)
		MesS						: REAL ; (* (kVA)Total Apparent power		       				*)
		MesCosPhi					: REAL ; (* (NA) Power factor                       			*)
		MesP1						: REAL ; (* (kW) Active Power Phase 1               			*)
		MesP2						: REAL ; (* (kW) Active Power Phase 2               			*)
		MesP3						: REAL ; (* (kW) Active Power phase 3               			*)
		MesQ1						: REAL ; (* (kVAr)Reactive Power Phase 1            			*)
		MesQ2						: REAL ; (* (kVAr)Reactive Power Phase 2            			*)
		MesQ3						: REAL ; (* (kVAr)Reactive Power Phase 3            			*)
		MesS1						: REAL ; (* (kVA) Total Apparent power Phase 1      			*)
		MesS2						: REAL ; (* (kVA) Total Apparent power Phase 2      			*)
		MesS3						: REAL ; (* (kVA) Total Apparent power Phase 3      			*)
		MesEActCons					: REAL ; (* (kWh) Recieved active energy            			*)
		MesEReactCons				: REAL ; (* (kVArh) 	Recieved reactive energy       			*)
		MesEActProd					: REAL ; (* (kWh) Delivered active energy           			*)
		MesEReactProd				: REAL ; (* (kVArh) 	Delivered reactive energy	   			*)
		MesI						: REAL ; (* (A) Mean AC current                     			*)
		MesV						: REAL ; (* (V) Mean Simple Phase AC Voltage        			*)
		MesU						: REAL ; (* (V) Mean Phase - Phase  AC Voltage      			*)
		MesCosPhi1                  : REAL ; (* (NA) Total Power Factor Phase 1         			*)
		MesCosPhi2                  : REAL ; (* (NA) Total Power Factor Phase 2         			*)
		MesCosPhi3                  : REAL ; (* (NA) Total Power Factor Phase 3         			*)
		MesTanPhi					: REAL ; (* (NA) Total Tangeante phi                			*)

		MesAlarmCom					: BOOL ;  		 (* (NA) Communication Error with I35 module    *)
		MesCP_Read					: BOOL := TRUE ; (* (NA) Cal: Read FUNCTION enable 				*)
		                                                                                        	
		MesAlarmCode				: WORD ; (* (NA) Internal Akuo Alarm Code			   			*)
		MesWarningCode				: WORD ; (* (NA) Internal Akuo Warning Code			  			*)
END_STRUCT
END_TYPE

// ---- 01_Equipement_Library/Operation Meter/PM_PM800.TcDUT
TYPE PM_PM800 :
STRUCT
	MesData 					: PM;
	
	MesTHD1 			: REAL;	(* Total Harmonic Distortion Phase 1, Adr 1199 *)
	MesTHD2 			: REAL;	(* Total Harmonic Distortion Phase 2, Adr 1200 *)
	MesTHD3 			: REAL;	(* Total Harmonic Distortion Phase 3, Adr 1201 *)
	MesTHD1N 			: REAL;	(* Total Harmonic Distortion Phase 1 - Neutre, Adr 1206 *)
	MesTHD2N 			: REAL;	(* Total Harmonic Distortion Phase 2 - Neutre, Adr 1207 *)
	MesTHD3N 			: REAL;	(* Total Harmonic Distortion Phase 3 - Neutre, Adr 1208 *)
END_STRUCT
END_TYPE

// ---- 01_Equipement_Library/Operation Meter/PM_Q100.TcDUT
TYPE PM_Q100 :
STRUCT
	//Device Status 
	MesState1		: WORD ;	(* Bit0: 1=Decide OK, Bit2: 0=Battery OK, Bit4:	1=SD card error, Bit8: 1= Parameter load is in progress, Bit10: 1=	parameter check is in progress, Bit12: 1=Parameter ativation is in progress *)
	MesState2		: WORD;		(* Bit0:	1= rotation is clockwis	*)
	                            
	MesData			: PM;       (**)
                                
	MesVN			: REAL;		(*  (V) Voltage neutral conductor  *)
	CalTanPhi		: REAL;		(*  (NA) TanPhi                    *)
	MesCosPhiA		: REAL;		(*  (NA) Active power factor a     *)
	MesCosPhiB		: REAL;		(*  (NA) Active power factor b     *)
	MesCosPhiC		: REAL;		(*  (NA) Active power factor c     *)
	MesCosPhi		: REAL;		(*  (NA) Active power factor       *)
	MesEPerPulse	: REAL;		(*  (Wh, VArh, VAh per pulse) COnversion factor of counter pulses into energy values    *)
	                            
	MesEac1_dmd		: REAL;		(* Active energy based on active power Pa Demand	Counter  *)
	MesEac2_dmd		: REAL;		(* Active energy based on active power Pb Demand	Counter  *)
	MesEac3_dmd		: REAL;		(* Active energy based on active power Pc Demand Counter     *)
	MesEac_dmd		: REAL;		(* Active energy based on active power Pa Demand Counter     *)
								                                                             
	MesEac1_sup		: REAL;		(* Active energy based on active power Pa Supply Counter     *)
	MesEac2_sup		: REAL;		(* Active energy based on active power Pb Supply Counter     *)
	MesEac3_sup		: REAL;		(* Active energy based on active power Pc Supply Counter     *)
	MesEac_sup		: REAL;		(* Active energy based on active power P Supply Counter      *)
								                                                                   
	MesEreac1_cap	: REAL;		(* Reactive energy based on reactive power Qa capacitive Counter   *)
	MesEreac2_cap	: REAL;		(* Reactive energy based on reactive power Qb capacitive Counter   *)
	MesEreac3_cap	: REAL;		(* Reactive energy based on reactive power Qc capacitive Counter   *)
	MesEreac_cap	: REAL;		(* Reactive energy based on reactive power Q capacitive Counter    *)
								                                                                   
	MesEreac1_ind	: REAL;		(* Reactive energy based on reactive power Qa inductive Counter    *)
	MesEreac2_ind	: REAL;		(* Reactive energy based on reactive power Qb inductive Counter    *)
	MesEreac3_ind	: REAL;		(* Reactive energy based on reactive power Qc inductive Counter    *)
	MesEreac_ind	: REAL;		(* Reactive energy based on reactive power Q  inductive Counter    *)
								                                                                   
	CalEac1_dmd		: REAL;		(* Active energy based on active power Pa Demand         *)
	CalEac2_dmd		: REAL;		(* Active energy based on active power Pb Demand         *)
	CalEac3_dmd		: REAL;		(* Active energy based on active power Pc Demand         *)
	CalEac_dmd		: REAL;		(* Active energy based on active power Pa Demand         *)
								                                                         
	CalEac1_sup		: REAL;		(* Active energy based on active power Pa Supply         *)
	CalEac2_sup		: REAL;		(* Active energy based on active power Pb Supply         *)
	CalEac3_sup		: REAL;		(* Active energy based on active power Pc Supply         *)
	CalEac_sup		: REAL;		(* Active energy based on active power P Supply          *)
								                                                         
	CalEreac1_cap	: REAL;		(* Reactive energy based on reactive power Qa capacitive *)
	CalEreac2_cap	: REAL;		(* Reactive energy based on reactive power Qb capacitive *)
	CalEreac3_cap	: REAL;	    (* Reactive energy based on reactive power Qc capacitive *)
	CalEreac_cap	: REAL;	    (* Reactive energy based on reactive power Q capacitive  *)
								                                                         
	CalEreac1_ind	: REAL;	    (* Reactive energy based on reactive power Qa inductive  *)
	CalEreac2_ind	: REAL;	    (* Reactive energy based on reactive power Qb inductive  *)
	CalEreac3_ind	: REAL;	    (* Reactive energy based on reactive power Qc inductive  *)
	CalEreac_ind	: REAL;	    (* Reactive energy based on reactive power Q  inductive  *)
		
	MesAlarmCodeAkuo			: WORD;		(* Akuo Custom AlarmCode	*)
	MesWarningCodeAkuo			: WORD;		(* Akuo Custom WarningCode	*)
	
	

END_STRUCT
END_TYPE

// ---- 01_Equipement_Library/Operation Meter/PM_SicamQ100.TcDUT
///////////
// Structure For I35. Main Operating Data to be saved ( ex: OPC ) .  
//////////
TYPE PM_SicamQ100 :
STRUCT
	
	MesData					: PM ; 

	MesState1			: WORD ; 	(* Power meter state 1 *)
	MesState2			: WORD ; (* Power meter state 2 *)
	MesEac1_dmd			: REAL ; (* (kWh)Eac  *)
	MesEac2_dmd         : REAL ; (* (kWh)Eac  *)
	MesEac3_dmd         : REAL ; (* (kWh)Eac  *)
	MesEac_dmd          : REAL ; (* (kWh)Eac  *)
	MesEac1_sup         : REAL ; (* (kWh)Eac  *)
	MesEac2_sup         : REAL ; (* (kWh)Eac  *)
	MesEac3_sup         : REAL ; (* (kWh)Eac  *)
	MesEac_sup          : REAL ; (* (kWh)Eac  *)
	MesEreac1_ind       : REAL ; (* (kVArh)Power meter state 1 *)
	MesEreac2_ind       : REAL ; (* (kVArh)Power meter state 1 *)
	MesEreac3_ind       : REAL ; (* (kVArh)Power meter state 1 *)
	MesEreac_ind        : REAL ; (* (kVArh)Power meter state 1 *)
	MesEreac1_cap       : REAL ; (* (kVArh)Power meter state 1 *)
	MesEreac2_cap       : REAL ; (* (kVArh)Power meter state 1 *)
	MesEreac3_cap       : REAL ; (* (kVArh)Power meter state 1 *)
	MesEreac_cap        : REAL ; (* (kVArh)Power meter state 1 *)
	
	
	MesEPerPulse 			: REAL ; (* (kWh)Energy per pulse *)
	
	
	
	
	
	

END_STRUCT
END_TYPE

// ---- 01_Equipement_Library/Operation Meter/PM_Standard.TcDUT
///////////
// Structure For I35. Main Operating Data to be saved (ex: OPC).  
//////////
TYPE PM_Standard :
STRUCT
		MesData						: PM ; (* Object *) 
	
END_STRUCT
END_TYPE

// ---- 01_Equipement_Library/PCS/PCS.TcDUT
///////////
// Structure for CtrlPcs Jema .  
//////////
TYPE PCS :
STRUCT
// PCS Controller  Measures
	MesP 						: REAL;  		// (kW)  Active Power 
	MesQ 						: REAL;  		// (kVAr) Reactive Power
	MesPdc 						: REAL;  		// (kW)  DC Power 
	MesCosPhi 					: REAL;  		// (p.u) Power factor
	MesU 						: REAL;  		// (V) 	AC Voltage measure
	MesFreq						: REAL;			// (Hz) Main Bus Freq
	MesUdc 						: REAL;  		// (V) 	DC Voltage measure
	MesI 						: REAL; 		// (A) 	Total AC current 
	MesIdc 						: REAL; 		// (A) 	Total DC current from batteries (+ = discharge)
	MesState					: WORD;			// (NA) [P,H,B] Bit0: 1 = Not Available (AC or DC breaker open or AllAcContactorsOpened), Bit1: GridMode: 1=grid
	MesTemp						: REAL;			// (°C) Temperature sensor
	MesHumidity					: REAL;			// (%) Humidity sensor
	MesPrecharge				: BOOL;			// (NA) Precharge indicator      
	MesDcBreaker				: BOOL;			// (NA) Dc Breaker status      
	MesSoCLimitReached			: BOOL; 		// (NA) SoC limit reached
    MesAcBreaker				: BOOL; 		// (NA) Ac Breaker status
	MesHeartBeat				: WORD; 		// (NA) HeartBeat of the Inverter
	MesS_BatChargeMax			: REAL;			// (kVA) Max apparent power available for Charge based on load factor
	MesS_BatDischargeMax		: REAL;			// (kVA) Max apparent power available for discharge based on load factor
	MesNbPcsConnected			: UINT; 		// (NA) Number of online PCS 
	MesAtLeastOnePcsConnected	: BOOL; 		// (NA) At least one Pcs connected and not in alarm
	MesOpeFlag					: WORD;			// (NA) Operation flag from PCS
	MesWarning 					: BOOL; 		// (NA) PCS Controller general Warning 
	MesComAlarm					: BOOL; 		// (NA) PCS Controller Communication fault
	MesComWarning				: BOOL;			// (NA) PCS Controller Communication warning
	MesOnGrid 					: BOOL; 		// TRUE if AFE in ONgrid Mode.
	MesOffGrid 					: BOOL; 		// TRUE if AFE in Offgrid Mode.                 	
	MesFreqReg_Active			: BOOL; 		// (NA) Is the frequency regulation active : True = FreqReg Active
	MesUReg_Active				: BOOL; 		// (NA) Is the voltage regulation active : True = UReg Active
	MesSnom						: REAL; 		// (kW) Nominal power read on Controller
	MesAvailability				: REAL; 		// (%) Availability of the inverter
	MesAlarmCode				: WORD;			// (NA) Internal Akuo AlarmCode
	MesWarningCode				: WORD; 		// (NA) Internal Akuo WarningCode
	MesEventCode				: WORD;			// (NA) Internal Akuo EventCode
	OUT_CmdStop					: BOOL; 		// (NA) Stop  sent to the Controller
	OUT_CmdStart				: BOOL;			// (NA) Start sent to the Controller
	OUT_CmdStandby				: BOOL;			// (NA) Soft stop sent to the Controller
	OUT_CmdInvLocal				: BOOL;			// (NA) If true, INV is excluded from regulation
	OUT_CmdP					: BOOL;			// (NA) P setpoint is enabled
	OUT_CmdQ					: BOOL;			// (NA) Q setpoint is enabled
	OUT_CmdCosPhi				: BOOL;			// (NA) CosPhi setpoint is enabled
	OUT_CmdBlackStart			: BOOL;			// (NA) Blackstart order sent to the controller
	OUT_CmdFreqregMode			: BOOL;			// (NA) Frequency regulation mode sent to the controller
	OUT_CmdUregMode				: BOOL;			// (NA) Voltage regulation mode sent to the controller
	OUT_CmdMicroCyclingMode		: BOOL;			// (NA) MicroCycling is active
	OUT_CmdGridMode				: BOOL;			// (NA) Mode of the PCS :  FALSE = Grid Feeder, TRUE = Grid Former
	OUT_CmdOpenAc				: BOOL;			// (NA) Open AC breaker order sent to controller
	OUT_CmdOpenDc				: BOOL;			// (NA) Open DC breaker order sent to controller
	OUT_SetptP					: REAL; 		// (kW) Active power setpoint 
	OUT_SetptPMax				: REAL;			// (kW) Upper range of the Active Power setpoint
	OUT_SetptPMin				: REAL;			// (kW) Lower range of the Active Power setpoint
	OUT_SetptQ					: REAL; 		// (kVAr) Reactive power setpoint 
	OUT_SetptQMax				: REAL;			// (kVAr) Upper range of the Reactive Power setpoint
	OUT_SetptQMin				: REAL;			// (kVAr) Lower range of the Reactive Power setpoint
	OUT_SetptCosPhi				: REAL;			// (NA) CosPhi setpoint
	OUT_MesV					: REAL;			// (V) Measure of the voltage sent to the Inverter for its regulation
	OUT_SetptV					: REAL;			// (V) Setpoint of the voltage sent to the Inverter for the OffGrid Mode
	OUT_SetptF					: REAL;			// (Hz) Setpoint of the frequency sent to the Inverter for the OffGrid Mode

	MesCP_Read					: BOOL := TRUE;	// (NA) CP to read values from PCS
	MesCP_Write					: BOOL := TRUE;	// (NA) CP to write values from PCS
	
END_STRUCT
END_TYPE

// ---- 01_Equipement_Library/PCS/PowerCol_Jema.TcDUT
///////////
// Structure For Jema Module 
//////////
TYPE PowerCol_Jema :
STRUCT
		MesPac 				: REAL; 		(* (kW) Active Power output (AC) of PCS										*)
		MesQac 				: REAL; 		(* (kVAr) Reactive AC Power Produced by PCS                                 *)
		MesPdc				: REAL ; 		(* (kW) DC Power .                                                          *)
		MesCosPhi 			: REAL;  		(* (p.u) Power factor                                                       *)
		MesFreq				: REAL ; 		(* (Hz) Frequency                                                           *)
		MesU 				: REAL;  		(* (V) AC Voltage measure                                                   *)
		MesUdc 				: REAL;  		(* (V) DC Voltage measure                                                   *)
		MesI 				: REAL; 		(* (A) Total AC current                                                     *)
		MesI1				: REAL ; 		(* (A) Phase 1 AC Current                                                   *)
		MesI2				: REAL ;        (* (A) Phase 2 AC Current                                                   *)
		MesI3				: REAL ;        (* (A) Phase 3 AC Current                                                   *)
		MesIdc 				: REAL; 		(* (A) Total DC current from batteries (+ = discharge)                      *)
		MesAcSwitchClosed	: BOOL ; 		(* (NA) Position of the AC Switch : True = Switch closed                    *)
		MesTempControl      : REAL ; 		(* (°C) Temperature of control card                                         *)
		MesTempPowerUnit    : REAL ;		(* (°C) Temperature of Power Unit                                           *)
		MesTempCabinet      : REAL ; 		(* (°C) Cabinet temperature                                                 *)
		MesRegAlarm0        : WORD ; 		(* Alarm Word of PCS                                                        *)
		MesRegAlarm1        : WORD ; 		(* Alarm Word of PCS                                                        *)
		MesRegAlarm2        : WORD ; 		(* Alarm Word of PCS                                                        *)
		MesRegAlarm3        : WORD ;  		(* Alarm Word of PCS                                                        *)
		MesRegAlarm4        : WORD ;  		(* Alarm Word of PCS                                                        *)
		MesDeratingWord		: WORD ;		(* Derating word of PCS                                                     *)
		MesHeartbit			: REAL ;		(* Heartbit                                                                 *)
		MesDoorOpened		: BOOL ; 		(* PCS Door is opened .                                                     *)
		MesMaster			: BOOL ; 		(* Power column is master ( stop in last ) .                                *)
		
		MesJemaAlarms		: PowerCol_Jema_Alarms;	(* Object *)

		
			

END_STRUCT
END_TYPE

// ALARM WORD SUB-EQUIPEMNT 
(*
//RegAlarm0
	FB_AlarmCodeManager
(
		bAlarm0			:= ,// I1_Alm      
 		bAlarm1			:= ,// I2_Alm      					   
		bAlarm2			:= ,// I3_Alm                               
		bAlarm3			:= ,// Vdc_High_Alm                         
		bAlarm4			:= ,// Vdc_Low_Alm                          
		bAlarm5			:= ,//                                      
		bAlarm6			:= ,// U12_High_Alm                         
		bAlarm7			:= ,// U12_Low_Alm                          
		bAlarm8			:= ,// U23_High_Alm                         
		bAlarm9			:= ,// U23_Low_Alm                          
		bAlarm10		:= ,// U31_High_Alm                         
		bAlarm11		:= ,// U31_Low_Alm                          
		bAlarm12		:= ,// Vd_High_Alm 						
		bAlarm13		:= ,// Vd_Low_Alm                           
		bAlarm14		:= ,// Vdc_Neg                              
		bAlarm15		:= ,//                                  
		wAlarmCode		=> 				
);   
//RegAlarm1
	FB_AlarmCodeManager
(
		bAlarm0			:= ,// U1223_Unbalance 
 		bAlarm1			:= ,// U2331_Unbalance 				   
		bAlarm2			:= ,// U3112_Unbalance                           
		bAlarm3			:= ,// InvertedPhase                             
		bAlarm4			:= ,// I12_Unbalance                             
		bAlarm5			:= ,// I23_Unbalance                             
		bAlarm6			:= ,// I31_Unbalance                             
		bAlarm7			:= ,// CouplingTimeout                           
		bAlarm8			:= ,// F_High                                    
		bAlarm9			:= ,// F_Low                                     
		bAlarm10		:= ,//                                           
		bAlarm11		:= ,// SPD Failure                               
		bAlarm12		:= ,// PcbOverTemp     					
		bAlarm13		:= ,// HeatsinkOverTemp                          
		bAlarm14		:= ,//                                           
		bAlarm15		:= ,// OvertempHyst                            
		wAlarmCode		=> 				
);   

	FB_AlarmCodeManager
(
		bAlarm0			:= ,//                   
 		bAlarm1			:= ,//                   			   
		bAlarm2			:= ,//                                        
		bAlarm3			:= ,//                                        
		bAlarm4			:= ,// GridCbOpened                           
		bAlarm5			:= ,// GridCbTrip                             
		bAlarm6			:= ,//                                        
		bAlarm7			:= ,//                                        
		bAlarm8			:= ,// GridContactFail                        
		bAlarm9			:= ,// DoorOpened                             
		bAlarm10		:= ,//                                        
		bAlarm11		:= ,//                                        
		bAlarm12		:= ,// VdcPrechargewrong 				
		bAlarm13		:= ,//                                        
		bAlarm14		:= ,// OverVoltHyst                           
		bAlarm15		:= ,// IdcMax                              
		wAlarmCode		=> 				
);   

	FB_AlarmCodeManager
(
		bAlarm0			:= ,// SKIIP1         
 		bAlarm1			:= ,// SKIIP2         	   
		bAlarm2			:= ,// SKIIP3                        
		bAlarm3			:= ,// SIIP_OT                       
		bAlarm4			:= ,// IMax                          
		bAlarm5			:= ,// EmergencyStop                 
		bAlarm6			:= ,// FPGA_WdogTrip                 
		bAlarm7			:= ,// StopEverything                
		bAlarm8			:= ,// ImdWarning                    
		bAlarm9			:= ,// ImdFault                      
		bAlarm10		:= ,//                               
		bAlarm11		:= ,// CoilOverTemp                  
		bAlarm12		:= ,//                		
		bAlarm13		:= ,// AlrmGrp1_Curr                 
		bAlarm14		:= ,// AlrmGrp2_Curr                 
		bAlarm15		:= ,// ShortCircuit_DC            
		wAlarmCode		=> 				
);   

	FB_AlarmCodeManager
(
		bAlarm0			:= ,//               
 		bAlarm1			:= ,//               	   
		bAlarm2			:= ,//                                
		bAlarm3			:= ,// PowerUnbalance                 
		bAlarm4			:= ,// Overpower                      
		bAlarm5			:= ,// IOutRMS                        
		bAlarm6			:= ,//                                
		bAlarm7			:= ,//                                
		bAlarm8			:= ,//                                
		bAlarm9			:= ,//                                
		bAlarm10		:= ,//                                
		bAlarm11		:= ,//                                
		bAlarm12		:= ,//               		
		bAlarm13		:= ,//                                
		bAlarm14		:= ,//                                
		bAlarm15		:= ,//                             
		wAlarmCode		=> 				
);   








*)

// ---- 01_Equipement_Library/PCS/PowerCol_Jema_Alarms.TcDUT
TYPE PowerCol_Jema_Alarms :
STRUCT

// ALARM0 bAlarm1
		MesI1_Alm			: BOOL; //I1_Alm
		MesI2_Alm			: BOOL; //I2_Alm
		MesI3_Alm			: BOOL; //I3_Alm
		MesVdc_High_Alm		: BOOL; //Vdc_High_Alm
		MesVdc_Low_Alm		: BOOL; //Vdc_Low_Alm
		                            // 
		MesU12_High_Alm		: BOOL; //U12_High_Alm
		MesU12_Low_Alm		: BOOL; //U12_Low_Alm
		MesU23_High_Alm		: BOOL; //U23_High_Alm
		MesU23_Low_Alm		: BOOL; //U23_Low_Alm
		MesU31_High_Alm		: BOOL; //U31_High_Alm
		MesU31_Low_Alm		: BOOL; //U31_Low_Alm
		MesVd_High_Alm		: BOOL; //Vd_High_Alm
		MesVd_Low_Alm		: BOOL; //Vd_Low_Alm
		MesVdc_Neg			: BOOL; //Vdc_Neg
		                            //
									//wAlarmCode
		
// ALARM1 bAlarm1
		MesU1223_Unbalance	: BOOL;//U1223_Unbalance
		MesU2331_Unbalance	: BOOL;//U2331_Unbalance
		MesU3112_Unbalance	: BOOL;//U3112_Unbalance
		MesInvertedPhase	: BOOL;//InvertedPhase
		MesI12_Unbalance	: BOOL;//I12_Unbalance
		MesI23_Unbalance	: BOOL;//I23_Unbalance
		MesI31_Unbalance	: BOOL;//I31_Unbalance
		MesCouplingTimeout	: BOOL;//CouplingTimeout
		MesF_High			: BOOL;//F_High
		MesF_Low			: BOOL;//F_Low
		//MesGrndFault		: BOOL;//GrndFault
		MesVaristor			: BOOL;//SPD Failure
		MesPcbOverTemp		: BOOL;//PcbOverTemp
		MesHeatsinkOverTemp	: BOOL;//HeatsinkOverTemp
		                           // :
		MesOvertempHyst		: BOOL;//OvertempHyst
		//wAlarmCode
// ALARM2 bAlarm1
								   // :
                                   // :
                                   // :
                                   // :
		MesGridCbOpened		: BOOL;//GridCbOpened
		MesGridCbTrip		: BOOL;//GridCbTrip
//		MesPanelContactFail	: BOOL;//PanelContactFail 
		                           // :
		MesGridContactFail	: BOOL;//GridContactFail 
		MesDoorOpened		: BOOL;//DoorOpened 
		                           // :
		                           // :
		MesVdcPrechargewrong: BOOL;//VdcPrechargewrong 
		                           // :
		MesOverVoltHyst		: BOOL;//OverVoltHyst 
		MesIdcMax			: BOOL;//IdcMax 
		//wAlarmCode
		
//ALARM3   bAlarm1                         
		MesSKIIP1			: BOOL; //SKIIP1
		MesSKIIP2			: BOOL; //SKIIP2
		MesSKIIP3			: BOOL; //SKIIP3
		MesSKIIP_OT			: BOOL; //SIIP_OT
		MesIMax				: BOOL; //IMax
		MesEmergencyStop	: BOOL; //EmergencyStop
		MesFPGA_WdogTrip	: BOOL; //FPGA_WdogTrip
		MesStopEverything	: BOOL; //StopEverything
		MesImdWarning		: BOOL; //ImdWarning
		MesImdFault			: BOOL; //ImdFault
		                            // :
		MesCoilOverTemp		: BOOL; //CoilOverTemp
		                            // :
		MesAlrmGrp1_Curr	: BOOL; //AlrmGrp1_Curr
		MesAlrmGrp2_Curr	: BOOL; //AlrmGrp2_Curr
		MesShortCircuit_DC	: BOOL; //ShortCircuit_DC
		//wAlarmCode
// ALARM4 bAlarm1
		//MesBatError			: BOOL;//BatError
		//MesBatCtlStop		: BOOL;//BatCtlStop
		//MesBatComErrors		: BOOL;//BatComErrors
		MesPowerUnbalance	: BOOL;//PowerUnbalance
		MesOverpower		: BOOL;//Overpower
		MesIOutRMS			: BOOL ; // IOutRMS
		//wAlarmCode
		
END_STRUCT
END_TYPE

// ---- 01_Equipement_Library/ProtectRelay/ProtectRelay.TcDUT
///////////
// Structure For I35. Main Operating Data to be saved (ex: OPC).  
//////////
TYPE ProtectRelay :
STRUCT
		MesI1						: REAL ; 			(* (A) Maximal Current measured before fault on phase 1*)
		MesI2						: REAL ;			(* (A) Maximal Current measured before fault on phase 2*)
		MesI3						: REAL ;			(* (A) Maximal Current measured before fault on phase 3*)
		MesI0						: REAL ; 			(*(A) Measured  maximal residual current               *)
		MesI						: REAL ;			(*(A) Phase current value (averaged)               	   *)
		                                        		                                                    
		MesFreq						: REAL ;			(* (Hz) Frequency measured                             *)
		                                        		                                                    
		MesImax1					: REAL ; 			(* (A) AC Max current during Fault phase 1             *)
		MesImax2                    : REAL ; 			(* (A) AC Max current during Fault phase 2             *)
		MesImax3                    : REAL ; 			(* (A) AC Max current during Fault phase 3		       *)
		MesImax0                    : REAL ; 			(* (A) AC Max residual current during Fault	           *)
		
		MesTripped                  : BOOL ;            (* Trip Synthesis *)                                        		                                                    
		MesAlarmCom					: BOOL ;			(* Communication Error with Sepam                      *)
                                                		                                                   
		MesAlarmTCS					: BOOL ; 			(* TCS in fault. RPN can not trip anymore              *)
		MesAlarmImax				: BOOL ; 			(* Imax alarm, ANSI Trip 50, 51 , 50G, 51G Synthesis                                       *)
		MesAlarmUmin				: BOOL ;			(* Short GTE Fault                                     *)
		MesAlarmUmin_Long			: BOOL ;			(* Long GTE FAULT                                      *)
      	MesAlarm_GTE3Time			: BOOL ; ;			(* 3 GTE FAULT   in 30 minutes                                   *)
		MesU12                      : REAL ;            (* (V) Voltage between phase 2 and phase 1 *)
		MesU23                      : REAL ;            (* (V) Voltage between phase 3 and phase 2 *)     
		MesU31                      : REAL ;            (* (V) Voltage between phase 1 and phase 3 *)                                                                                              
		
		MesWatchdog	                : BOOL ;            (* Watchdog *) 

		MesCP_Read					: BOOL := FALSE;	(* Cal Read function enable                            *)
		MesCP_Write					: BOOL := FALSE;	(* Cal Write function enable                           *)
		                                                                                                     
		MesAlarmCode				: WORD ; 			(* (NA) Internal Akuo AlarmCode                        *)
		MesWarningCode				: WORD ; 			(* (NA) Internal Akuo WarningCode                      *)
		MesEventCode				: WORD ; 			(* (NA) Internal Akuo EventCode		                   *)
		
END_STRUCT
END_TYPE

// ---- 01_Equipement_Library/ProtectRelay/ProtectRelay_Flair23DM.TcDUT
TYPE ProtectRelay_Flair23DM :
STRUCT
		MesData						: ProtectRelay;		(* (NA) Protection relay			  *)
               
		MesV1						: REAL ; 			(* (V) Output Phase Voltage Phase 1   *)
		MesV2						: REAL ; 			(* (V) Output Phase Voltage Phase 2   *)
		MesV3						: REAL ; 			(* (V) Output Phase Voltage Phase 3   *)
		MesV0						: REAL ; 		    (* (V) Residual Voltage				  *)
		
		MesStateCom					: BOOL ; 			(* (NA) False=NotOK. Device did not respond successfully to most recent read/write request. True= Device is responding normally *)
	  	
		ControlWord					: WORD ; 			(* (NA) Control Word				 *)
	   	StatusWord					: WORD ; 			(* (NA) Status Word                  *)
		CalToggleWrite				: BOOL ;			(* (NA) True := read authorised      *)
		CalToggleRead				: BOOL ;			(* (NA) True := Write authorised     *)
		       
END_STRUCT
END_TYPE

// ---- 01_Equipement_Library/ProtectRelay/ProtectRelay_NSXCB.TcDUT
TYPE ProtectRelay_NSXCB :
STRUCT
		MesData						: ProtectRelay;			(* (NA) Protection relay				*)
               
		MesStatCom					: BOOL; 				(* (NA) False:=.:NotOK.Device did notrespond successfullyto most recentread orwrite request, TRUE := Device is responding normally *)
	                                        				
		MesMaxFreq					: REAL; 				(* (Hz) Frequence max					*)
		                                    				
		MesP1						: REAL; 				(* (kW) Active poweron phase 1 (P1) 	*)
		MesP2						: REAL; 				(* (kW) Active poweron phase 2 (P1) 	*)
		MesP3						: REAL; 				(* (kW) Active poweron phase 3 (P1) 	*)
        MesPtot						: REAL; 				(* (kW) Total active power(Ptot)    	*)
		                                    				
		MesQ1						: REAL; 				(* (kvar) Reactive poweron phase 1 (Q1) *)
		MesQ2						: REAL; 				(* (kvar) Reactive poweron phase 1 (Q2) *)
		MesQ3						: REAL; 				(* (kvar) Reactive poweron phase 1 (Q3) *)
		MesQtot						: REAL; 				(* (kvar) Total reactive power(Qtot)    *)
		                                    				
		MesS1						: REAL; 				(* (kVA) Apparent power on phase 1 		*)
		MesS2						: REAL; 				(* (kVA) Apparent power on phase 2 		*)
		MesS3						: REAL; 				(* (kVA) Apparent power on phase 3 		*)
		MesStot						: REAL;					(* (kVA) Total apparentpower(Stot) 		*)
		                                    				
		MesEAct						: REAL; 				(* (Wh)  Active energy       			*)
		MesEReact					: REAL; 				(* (VArh)Reactive energy		   		*)
		                                    				
		MesCosPhi1					: REAL; 				(* (pu) Power factor on phase 1  		*)
		MesCosPhi2					: REAL; 				(* (pu) Power factor on phase 2  		*) 	
		MesCosPhi3					: REAL; 				(* (pu) Power factor on phase 3  		*)
		MesCosPhi					: REAL; 				(* (pu) Power factor on phase Tot		*)
		
